// TwinCAT 3 PLC project AnalyticsPLC
// ProgramVersion: 3.1.4026.16
// libraries:
//   Tc2_EtherCAT, * (Beckhoff Automation GmbH)
//   Tc2_Standard, * (Beckhoff Automation GmbH)
//   Tc2_System, * (Beckhoff Automation GmbH)
//   Tc2_Utilities, * (Beckhoff Automation GmbH)
//   Tc3_Analytics, * (Beckhoff Automation GmbH)
//   Tc3_AnalyticsCommunication, * (Beckhoff Automation GmbH)
//   Tc3_EventLogger, * (Beckhoff Automation GmbH)
// project tree:
//   / AnalyticsTask.TcTTO, AnalyticsTask_C1.TcTTO, PlcTask.TcTTO
//   DUTs/Analytics/ Color.TcDUT, E_AnalysisComponents.TcDUT, E_DataSourceContext.TcDUT, E_DataSourceState.TcDUT, E_DTType.TcDUT, E_ScopeCommand.TcDUT, E_VirtualInput.TcDUT, Shapes.TcDUT, ST_AnalysisReset.TcDUT
//   DUTs/Analytics/HMI/Controls/ ST_HMI_C1_Ctrl1_Production_Quantity_Analysis.TcDUT, ST_HMI_C1_Ctrl2_OEE_Trend_Line.TcDUT, ST_HMI_C1_Ctrl3_Productivity_Interval.TcDUT, ST_HMI_C1_Ctrl4_Overall_Equipment_Effectiveness_OEE.TcDUT
//   DUTs/Analytics/HMI/DataSourcePage/ E_SourceType.TcDUT, ST_HMI_DataSourceConfig.TcDUT, ST_HMI_DataSourceCtrl.TcDUT, ST_HMI_DataSourceHist.TcDUT, ST_HMI_DataSourceHistInfo.TcDUT, ST_HMI_DataSourceHistRecordInfo.TcDUT, ST_HMI_InputSource.TcDUT, ST_HMI_InputSourceCtrl.TcDUT
//   DUTs/Analytics/HMI/ ST_HMI_C1_OEE_Status.TcDUT, ST_HMI_MapItem.TcDUT, ST_KeyValuePair.TcDUT
//   DUTs/Analytics/Results/ ST_Results.TcDUT
//   DUTs/Analytics/Sources/ ST_T1_Inputs.TcDUT
//   GVLs/ Analytics.TcGVL, AnalyticsHMI.TcGVL
//   POUs/Analytics/Analysis/ FB_Analysis.TcPOU
//   POUs/Analytics/Analysis/Networks/N01 OEEStatus/ FB_N1_OEEStatus.TcPOU
//   POUs/Analytics/Analysis/Networks/N01 OEEStatus/Modules/ FB_N1_M1_OverallEquipmentEffectivenessOEE.TcPOU, FB_N1_M2_ProductionModeTimingAnalysis.TcPOU, FB_N1_M3_OEETrendLine.TcPOU, FB_N1_M4_ProductionQuantityAnalysis.TcPOU, FB_N1_M5_ProductivityInterval.TcPOU
//   POUs/Analytics/ MAIN_Analytics.TcPOU, MAIN_Analytics_C1.TcPOU
//   POUs/Analytics/Sources/T1_InputSource/ FB_T1_InputSource.TcPOU
//   POUs/Analytics/Sources/[Interfaces]/ I_InputSource.TcIO, I_InputSourceHistorical.TcIO
//   POUs/Analytics/VirtualInputSources/C1_Configuration_1/ FB_V1_C1_VirtualInputSource.TcPOU
//   POUs/Analytics/VirtualInputSources/[Interfaces]/ I_V1_VirtualInputSource.TcIO, I_VirtualInputSource.TcIO
//   POUs/Analytics/[Helper]/Common/ FB_DataBuffer.TcPOU, FB_GetSampleIndex.TcPOU, FB_TcMessageSuccess.TcPOU, F_ANY_Negation.TcPOU, F_ARRAY_To_LREAL_ARRAY.TcPOU, F_HasContext.TcPOU, F_ToANY.TcPOU
//   POUs/Analytics/[Helper]/Convert Timestamp/ F_AlyTimestampToDCTimestruct.TcPOU, F_AlyTimestampToFileTime.TcPOU, F_AlyTimestampToLocalTime.TcPOU, F_DCTimestructToFileTime.TcPOU, F_FileTimeToDCTimestruct.TcPOU, F_RawTimeToDCTimestruct.TcPOU
//   POUs/Analytics/[Helper]/ F_SampleTimeCheck.TcPOU
//   POUs/ MAIN.TcPOU
// (motion and I/O tree: see PLC project unbenannt1)
// real-time tasks:
//   TASK PlcTask: cycle T#10ms, priority 20, ADS port 350
//   TASK PlcTask1: cycle T#10ms, priority 21, ADS port 351
//   TASK AnalyticsTask: cycle T#10ms, priority 1, ADS port 352
//   TASK AnalyticsTask_C1: cycle T#10ms, priority 22, ADS port 353
// variable links:

CONFIGURATION AnalyticsPLC
    RESOURCE PLC ON TwinCAT3
        TASK AnalyticsTask(INTERVAL := T#10ms, PRIORITY := 1);
        TASK AnalyticsTask_C1(INTERVAL := T#10ms, PRIORITY := 22);
        TASK PlcTask(INTERVAL := T#10ms, PRIORITY := 21);
        PROGRAM MAIN_Analytics WITH AnalyticsTask : MAIN_Analytics;
        PROGRAM MAIN_Analytics_C1 WITH AnalyticsTask_C1 : MAIN_Analytics_C1;
        PROGRAM MAIN WITH PlcTask : MAIN;
    END_RESOURCE
END_CONFIGURATION

// ---- DUTs/Analytics/Color.TcDUT
{attribute 'qualified_only'}
{attribute 'strict'}
TYPE Color : 
(
	White := 0,
	Black,
	Red,
	Green,
	Blue
) ;
END_TYPE

// ---- DUTs/Analytics/E_AnalysisComponents.TcDUT
{attribute 'qualified_only'}
{attribute 'strict'}
TYPE E_AnalysisComponents : 
(
	All := -1,
	N1_OEEStatus := 0,
	N1_M1_OverallEquipmentEffectivenessOEE := 1,
	N1_M2_ProductionModeTimingAnalysis := 2,
	N1_M3_OEETrendLine := 3,
	N1_M4_ProductionQuantityAnalysis := 4,
	N1_M5_ProductivityInterval := 5,
	V1_VirtualInputSource := 6
) ;
END_TYPE

// ---- DUTs/Analytics/E_DataSourceContext.TcDUT
{attribute 'qualified_only'}
TYPE E_DataSourceContext : 
(
	eContext_No := 0, //
	eContext_Unknown := 2#0000_0000_0000_0001_0000_0000_0000_0000, //Unknown - All contexts allowed
	eContext_10000 := 2#0000_0000_0000_0010_0000_0000_0000_0000, //10000 µs
	eContext_Reserve1 := 2#0000_0000_0000_0100_0000_0000_0000_0000, //Reserve
	eContext_Reserve2 := 2#0000_0000_0000_1000_0000_0000_0000_0000, //Reserve
	eContext_Reserve3 := 2#0000_0000_0001_0000_0000_0000_0000_0000, //Reserve
	eContext_Reserve4 := 2#0000_0000_0010_0000_0000_0000_0000_0000, //Reserve
	eContext_Reserve5 := 2#0000_0000_0100_0000_0000_0000_0000_0000, //Reserve
	eContext_Reserve6 := 2#0000_0000_1000_0000_0000_0000_0000_0000, //Reserve
	eContext_Reserve7 := 2#0000_0001_0000_0000_0000_0000_0000_0000, //Reserve
	eContext_Reserve8 := 2#0000_0010_0000_0000_0000_0000_0000_0000, //Reserve
	eContext_Reserve9 := 2#0000_0100_0000_0000_0000_0000_0000_0000, //Reserve
	eContext_Reserve10 := 2#0000_1000_0000_0000_0000_0000_0000_0000, //Reserve
	eContext_Reserve11 := 2#0001_0000_0000_0000_0000_0000_0000_0000, //Reserve
	eContext_Reserve12 := 2#0010_0000_0000_0000_0000_0000_0000_0000, //Reserve
	eContext_Reserve13 := 2#0100_0000_0000_0000_0000_0000_0000_0000, //Reserve
	eContext_Reserve14 := 2#1000_0000_0000_0000_0000_0000_0000_0000 //Reserve
) DWORD;
END_TYPE

// ---- DUTs/Analytics/E_DataSourceState.TcDUT
{attribute 'qualified_only'}
{attribute 'strict'}
TYPE E_DataSourceState : 
(
	eUnknown := 0,
	eNotConnected,
	eReceiveData,
	eReceiveData_Cancel,
	eReceiveData_Pause,
	eError,
	eReady,
	eWaitForData
) ;
END_TYPE

// ---- DUTs/Analytics/E_DTType.TcDUT
{attribute 'qualified_only'}
{attribute 'strict'}
TYPE E_DTType : 
(
	NotInitialized := 0,
	BOOL_,
	BYTE_,
	WORD_,
	DWORD_,
	SINT_,
	USINT_,
	INT_,
	UINT_,
	DINT_,
	UDINT_,
	LINT_,
	ULINT_,
	REAL_,
	LREAL_,
	LWORD_
) ;
END_TYPE

// ---- DUTs/Analytics/E_ScopeCommand.TcDUT
{attribute 'qualified_only'}
{attribute 'strict'}
TYPE E_ScopeCommand : 
(
	eDefault := 0,
	ePause,
	eStop
) ;
END_TYPE

// ---- DUTs/Analytics/E_VirtualInput.TcDUT
{attribute 'qualified_only'}
TYPE E_VirtualInput : 
(
	eContext_No := 0, //
	eContext_V1_VirtualInputSource := 2#0000_0000_0000_0000_0000_0000_0000_0001, //VirtualInputSource
	eContext_Vn_Reserve1 := 2#0000_0000_0000_0000_0000_0000_0000_0010, //Reserve
	eContext_Vn_Reserve2 := 2#0000_0000_0000_0000_0000_0000_0000_0100, //Reserve
	eContext_Vn_Reserve3 := 2#0000_0000_0000_0000_0000_0000_0000_1000, //Reserve
	eContext_Vn_Reserve4 := 2#0000_0000_0000_0000_0000_0000_0001_0000, //Reserve
	eContext_Vn_Reserve5 := 2#0000_0000_0000_0000_0000_0000_0010_0000, //Reserve
	eContext_Vn_Reserve6 := 2#0000_0000_0000_0000_0000_0000_0100_0000, //Reserve
	eContext_Vn_Reserve7 := 2#0000_0000_0000_0000_0000_0000_1000_0000, //Reserve
	eContext_Vn_Reserve8 := 2#0000_0000_0000_0000_0000_0001_0000_0000, //Reserve
	eContext_Vn_Reserve9 := 2#0000_0000_0000_0000_0000_0010_0000_0000, //Reserve
	eContext_Vn_Reserve10 := 2#0000_0000_0000_0000_0000_0100_0000_0000, //Reserve
	eContext_Vn_Reserve11 := 2#0000_0000_0000_0000_0000_1000_0000_0000, //Reserve
	eContext_Vn_Reserve12 := 2#0000_0000_0000_0000_0001_0000_0000_0000, //Reserve
	eContext_Vn_Reserve13 := 2#0000_0000_0000_0000_0010_0000_0000_0000, //Reserve
	eContext_Vn_Reserve14 := 2#0000_0000_0000_0000_0100_0000_0000_0000, //Reserve
	eContext_Vn_Reserve15 := 2#0000_0000_0000_0000_1000_0000_0000_0000 //Reserve
) DWORD;
END_TYPE

// ---- DUTs/Analytics/HMI/Controls/ST_HMI_C1_Ctrl1_Production_Quantity_Analysis.TcDUT
TYPE ST_HMI_C1_Ctrl1_Production_Quantity_Analysis : 
STRUCT
	//Production Quantity Analysis
	bTrigReconfigure: BOOL;
	fM4_nCyclesElapsed: LREAL; //Elapsed (Values)
	fM4_nCyclesRemaining: LREAL; //Remaining (Values)
END_STRUCT
END_TYPE

// ---- DUTs/Analytics/HMI/Controls/ST_HMI_C1_Ctrl2_OEE_Trend_Line.TcDUT
TYPE ST_HMI_C1_Ctrl2_OEE_Trend_Line : 
STRUCT
	//OEE Trend Line
	bTrigReconfigure: BOOL;
	aM3_aTrendData: ARRAY [1..4] OF ARRAY [1..10080] OF LREAL; //Raw Data
	tM3_fbLastValue: DCTIMESTRUCT; //Last Value Timestamp
	nM3_nCountValues: UDINT; //Counted Values
	aM3_aChannelNames: ARRAY [0..3] OF STRING(255); //Display Names
END_STRUCT
END_TYPE

// ---- DUTs/Analytics/HMI/Controls/ST_HMI_C1_Ctrl3_Productivity_Interval.TcDUT
TYPE ST_HMI_C1_Ctrl3_Productivity_Interval : 
STRUCT
	//Productivity Interval
	bTrigReconfigure: BOOL;
	fM5_nProducedInInterval: LREAL; //Produced Pieces
	fM5_nRemainingInInterval: LREAL; //Remaining Pieces
	tM5_fbElapsedTime: ST_ALY_TimeSpan; //Elapsed Time
	tM5_fbRemainingTime: ST_ALY_TimeSpan; //Remaining Time
	fM5_fCurrentProductivity: LREAL; //Current Productivity
	fM5_fExpectedProductivity: LREAL; //Expected Productivity
END_STRUCT
END_TYPE

// ---- DUTs/Analytics/HMI/Controls/ST_HMI_C1_Ctrl4_Overall_Equipment_Effectiveness_OEE.TcDUT
TYPE ST_HMI_C1_Ctrl4_Overall_Equipment_Effectiveness_OEE : 
STRUCT
	//Overall Equipment Effectiveness (OEE)
	bTrigReconfigure: BOOL;
	fM1_fOEE: LREAL; //Overall equipment effectiveness (OEE)
	fM1_fAvailability: LREAL; //Availability
	fM1_fPerformance: LREAL; //Performance
	fM1_fQuality: LREAL; //Quality
	fM1_fThresholdLevelOkWarning: LREAL; //Level Ok / Warning
	fM1_fThresholdLevelWarningAlarm: LREAL; //Level Warning / Alarm
	eM1_eOeeClass: E_ALY_Classification_3Cls; //OEE Classification
END_STRUCT
END_TYPE

// ---- DUTs/Analytics/HMI/DataSourcePage/E_SourceType.TcDUT
{attribute 'qualified_only'}
{attribute 'strict'}
TYPE E_SourceType : 
(
	eLive := 0,
	eHistMQTT,
	eHistFile
) ;
END_TYPE

// ---- DUTs/Analytics/HMI/DataSourcePage/ST_HMI_DataSourceConfig.TcDUT
TYPE ST_HMI_DataSourceConfig : 
STRUCT
	nID: DINT;
	sDisplayName: WSTRING(80);
	eConfigType: E_SourceType;
	aInputSources: ARRAY [0..0] OF ST_HMI_InputSource;
END_STRUCT
END_TYPE

// ---- DUTs/Analytics/HMI/DataSourcePage/ST_HMI_DataSourceCtrl.TcDUT
TYPE ST_HMI_DataSourceCtrl : 
STRUCT
	nActiveConfigurationIdx: INT;
	
	aInputSourceCtrls: ARRAY [0..0] OF ST_HMI_InputSourceCtrl;
	
	bStart: BOOL;
	bCancel: BOOL;
	bPause: BOOL;
	bReset: BOOL;
	
	bUpdateRecordList: BOOL;
END_STRUCT
END_TYPE

// ---- DUTs/Analytics/HMI/DataSourcePage/ST_HMI_DataSourceHist.TcDUT
TYPE ST_HMI_DataSourceHist : 
STRUCT
	nCurrentRecordID: DINT;
	stSourceInfo: ST_HMI_DataSourceHistInfo;
	nRecordCount: DINT;
	aRecords: ARRAY [0..255] OF ST_HMI_DataSourceHistRecordInfo;
END_STRUCT
END_TYPE

// ---- DUTs/Analytics/HMI/DataSourcePage/ST_HMI_DataSourceHistInfo.TcDUT
TYPE ST_HMI_DataSourceHistInfo : 
STRUCT
	sSPGuid: GUID;
	sAlyFilePath: STRING(255);
	sSourceType: STRING(80);
	sTopic: STRING(255);
	sLayoutID: GUID;
END_STRUCT
END_TYPE

// ---- DUTs/Analytics/HMI/DataSourcePage/ST_HMI_DataSourceHistRecordInfo.TcDUT
TYPE ST_HMI_DataSourceHistRecordInfo : 
STRUCT
	nID: DINT;
	sName: WSTRING(80);
	sDisplayName: WSTRING(80);
	dtRecordStart: DCTIMESTRUCT;
	dtRecordEnd: DCTIMESTRUCT;
	dtSelectedRangeStart: DCTIMESTRUCT;
	dtSelectedRangeEnd: DCTIMESTRUCT;
END_STRUCT
END_TYPE

// ---- DUTs/Analytics/HMI/DataSourcePage/ST_HMI_InputSource.TcDUT
TYPE ST_HMI_InputSource : 
STRUCT
	nID: DINT;
	sDisplayName: WSTRING(80);
	
	sStreamSystemID: GUID;
	sTopic: STRING(255);
	
	eSourceType: E_SourceType;;
	eState: E_DataSourceState;;
	dtTimestamp: DCTIMESTRUCT;
	
	stHist: ST_HMI_DataSourceHist;
END_STRUCT
END_TYPE

// ---- DUTs/Analytics/HMI/DataSourcePage/ST_HMI_InputSourceCtrl.TcDUT
TYPE ST_HMI_InputSourceCtrl : 
STRUCT
	nActiveRecordIdx: INT;
	
	dtSelectedRangeStart: DCTIMESTRUCT;
	dtSelectedRangeEnd: DCTIMESTRUCT;
	
	bStart: BOOL;
	bCancel: BOOL;
	bPause: BOOL;
	bReset: BOOL;
END_STRUCT
END_TYPE

// ---- DUTs/Analytics/HMI/ST_HMI_C1_OEE_Status.TcDUT
TYPE ST_HMI_C1_OEE_Status : 
STRUCT
	stHMI_C1_Ctrl4_Overall_Equipment_Effectiveness_OEE: ST_HMI_C1_Ctrl4_Overall_Equipment_Effectiveness_OEE;
	
	stHMI_C1_Ctrl2_OEE_Trend_Line: ST_HMI_C1_Ctrl2_OEE_Trend_Line;
	
	stHMI_C1_Ctrl1_Production_Quantity_Analysis: ST_HMI_C1_Ctrl1_Production_Quantity_Analysis;
	
	stHMI_C1_Ctrl3_Productivity_Interval: ST_HMI_C1_Ctrl3_Productivity_Interval;
END_STRUCT
END_TYPE

// ---- DUTs/Analytics/HMI/ST_HMI_MapItem.TcDUT
TYPE ST_HMI_MapItem : 
STRUCT
	sName: WSTRING(127);
	sDescription: WSTRING(127);
	sPosition: WSTRING(127);
	nStatus: INT;
END_STRUCT
END_TYPE

// ---- DUTs/Analytics/HMI/ST_KeyValuePair.TcDUT
TYPE ST_KeyValuePair : 
STRUCT
	sKey: WSTRING(127);
	sValue: STRING(255);
END_STRUCT
END_TYPE

// ---- DUTs/Analytics/Results/ST_Results.TcDUT
TYPE ST_Results : 
STRUCT
END_STRUCT
END_TYPE

// ---- DUTs/Analytics/Shapes.TcDUT
{attribute 'qualified_only'}
{attribute 'strict'}
TYPE Shapes : 
(
	Rectangle := 0,
	Triangle,
	Pentagon,
	Hexagon,
	Circle
) ;
END_TYPE

// ---- DUTs/Analytics/Sources/ST_T1_Inputs.TcDUT
TYPE ST_T1_Inputs : 
STRUCT
	bGlobalVariables_bProductionMode: BOOL; //GlobalVariables.bProductionMode
	nGlobalVariables_lScheduledTime: LINT; //GlobalVariables.lScheduledTime
	nGlobalVariables_uProcessedCount: ULINT; //GlobalVariables.uProcessedCount
	nGlobalVariables_nVisuProductCommand: DINT; //GlobalVariables.nVisuProductCommand
	nGlobalVariables_uDefectiveCount: ULINT; //GlobalVariables.uDefectiveCount
	nGlobalVariables_lStartTime: LWORD; //GlobalVariables.lStartTime
	nGlobalVariables_lStopTime: LWORD; //GlobalVariables.lStopTime
	bGlobalVariables_bConfigure: BOOL; //GlobalVariables.bConfigure
	bGlobalVariables_bReset: BOOL; //GlobalVariables.bReset
	bGlobalVariables_bTest: BOOL; //GlobalVariables.bTest
	nGlobalVariables_uTotalCount: ULINT; //GlobalVariables.uTotalCount
END_STRUCT
END_TYPE

// ---- DUTs/Analytics/ST_AnalysisReset.TcDUT
TYPE ST_AnalysisReset : 
STRUCT
	eResetComponent: E_AnalysisComponents := E_AnalysisComponents.All;
	bResetExecute: BOOL;
END_STRUCT
END_TYPE

// ---- GVLs/Analytics.TcGVL
{attribute 'qualified_only'}
VAR_GLOBAL
	//DataSources
	//Live:
	fbT1_InputSource: FB_T1_InputSource;
	//Historical:
	//Empty:
	
	fbT1_IecCriticalSection: FB_IecCriticalSection;
	
	//Historical DataSource parameter
	nHistMaxInputBuffer: UDINT := 100;
	nHistMaxSampleCount: UDINT := 100;
	
	stReset: ST_AnalysisReset;
	
	//Scope ADS Push Target NetID
	sScopeServerNetID: T_AmsNetID := '10.123.65.55.1.1';
END_VAR

// ---- GVLs/AnalyticsHMI.TcGVL
{attribute 'qualified_only'}
VAR_GLOBAL
	//Switch between historical and live data
	stHMI_DataSourceCtrl: ST_HMI_DataSourceCtrl;
	stHMI_DataSourceConfig: ARRAY [0..0] OF ST_HMI_DataSourceConfig := [ 
																	( nID:= 1, sDisplayName:= "Configuration 1", eConfigType:= E_SourceType.eLive, 
																		aInputSources:= [ 
																			( nID:= 1, sDisplayName:= "1aa71777-6a15-92b4-38b4-ceb9ef9aa20f", sStreamSystemID:= STRING_TO_GUID('1aa71777-6a15-92b4-38b4-ceb9ef9aa20f'), 
																				sTopic:= 'PackMLDemo/PlcStream1', eSourceType:= E_SourceType.eLive, eState:= E_DataSourceState.eUnknown ) ] ) ];
	
	//Reset
	bN1_OEEStatus_Reset: BOOL;
	bN1_M1_OverallEquipmentEffectivenessOEE_Reset: BOOL;
	bN1_M2_ProductionModeTimingAnalysis_Reset: BOOL;
	bN1_M3_OEETrendLine_Reset: BOOL;
	bN1_M4_ProductionQuantityAnalysis_Reset: BOOL;
	bN1_M5_ProductivityInterval_Reset: BOOL;
	
	//Virtual Inputs
	bV1_bProductionMode: BOOL;
	nV1_lScheduledTime: LINT;
	nV1_uDefectiveCount: ULINT;
	nV1_lStartTime: LWORD;
	nV1_lStopTime: LWORD;
	bV1_bConfigure: BOOL;
	bV1_bReset: BOOL;
	bV1_bTest: BOOL;
	nV1_uTotalCount: ULINT;
	
	//HMI Structs
	stHMI_C1_OEE_Status: ST_HMI_C1_OEE_Status;
	
	//HMI Map Items
	aMapItems: ARRAY [0..0] OF ST_HMI_MapItem := [(sName:="1aa71777-6a15-92b4-38b4-ceb9ef9aa20f", sDescription:="", sPosition:="3 International Business Park, #05-07/08 Nordic European Centre, Singapore 609927", nStatus:= 0)];
END_VAR
VAR_GLOBAL CONSTANT
	nInstanceId: ULINT := 12860370723493188529;
END_VAR

// ---- POUs/Analytics/Sources/[Interfaces]/I_InputSource.TcIO
INTERFACE I_InputSource

METHOD AddClient : BOOL
VAR_OUTPUT
	nClientID: LWORD;
END_VAR
END_METHOD

METHOD Call : BOOL
END_METHOD

METHOD ClientDone : BOOL
VAR_INPUT
	nClientID: LWORD;
END_VAR
END_METHOD

METHOD GetData : BOOL
VAR_INPUT
	nElement: UDINT;
	pInputs: PVOID;
	nInputsSize: UDINT;
END_VAR
VAR_OUTPUT
	nTimestamp: ULINT;
	nContext: DWORD;
END_VAR
END_METHOD

METHOD NewDataAvailable : BOOL
VAR_INPUT
	nLastDataHandle: ULINT;
END_VAR
END_METHOD

PROPERTY eDataState : E_DataSourceState
GET
END_GET
END_PROPERTY

PROPERTY bReadNewData : BOOL
GET
END_GET
END_PROPERTY

PROPERTY nDataHandle : ULINT
GET
END_GET
END_PROPERTY

PROPERTY nElements : UDINT
GET
END_GET
END_PROPERTY

END_INTERFACE

// ---- POUs/Analytics/Sources/[Interfaces]/I_InputSourceHistorical.TcIO
INTERFACE I_InputSourceHistorical EXTENDS I_InputSource

METHOD HistoricalCtrl : BOOL
VAR_INPUT
	stCtrl: REFERENCE TO ST_HMI_InputSourceCtrl;
	stHistStreamInfo: REFERENCE TO ST_HMI_DataSourceHist;
	stRecordInfo: REFERENCE TO ST_HMI_DataSourceHistRecordInfo;
END_VAR
END_METHOD

METHOD UpdateRecordList : BOOL
VAR_INPUT
	sStreamSystemID: GUID;
	stHistStreamInfo: REFERENCE TO ST_HMI_DataSourceHist;
END_VAR
END_METHOD

PROPERTY bCtrlChanged : BOOL
GET
END_GET
END_PROPERTY

END_INTERFACE

// ---- POUs/Analytics/VirtualInputSources/[Interfaces]/I_V1_VirtualInputSource.TcIO
INTERFACE I_V1_VirtualInputSource EXTENDS I_VirtualInputSource

PROPERTY nV1_TimeLine : ULINT
GET
END_GET
END_PROPERTY

PROPERTY bV1_bProductionMode : BOOL
GET
END_GET
END_PROPERTY

PROPERTY nV1_lScheduledTime : LINT
GET
END_GET
END_PROPERTY

PROPERTY nV1_uDefectiveCount : ULINT
GET
END_GET
END_PROPERTY

PROPERTY nV1_lStartTime : LWORD
GET
END_GET
END_PROPERTY

PROPERTY nV1_lStopTime : LWORD
GET
END_GET
END_PROPERTY

PROPERTY bV1_bConfigure : BOOL
GET
END_GET
END_PROPERTY

PROPERTY bV1_bReset : BOOL
GET
END_GET
END_PROPERTY

PROPERTY bV1_bTest : BOOL
GET
END_GET
END_PROPERTY

PROPERTY nV1_uTotalCount : ULINT
GET
END_GET
END_PROPERTY

END_INTERFACE

// ---- POUs/Analytics/VirtualInputSources/[Interfaces]/I_VirtualInputSource.TcIO
INTERFACE I_VirtualInputSource

METHOD Done : BOOL
END_METHOD

METHOD NextData : BOOL
VAR_INPUT
	nMaxOversampling: UDINT;
END_VAR
END_METHOD

METHOD SourceSync : BOOL
END_METHOD

PROPERTY bEndOfData : BOOL
GET
END_GET
END_PROPERTY

PROPERTY dtTimestamp : DCTIMESTRUCT
GET
END_GET
END_PROPERTY

PROPERTY nContext : DWORD
GET
END_GET
END_PROPERTY

PROPERTY nDataHandle : ULINT
GET
END_GET
END_PROPERTY

PROPERTY tTimestamp : ULINT
GET
END_GET
END_PROPERTY

PROPERTY nMaxOversamplingFactor : UDINT
GET
END_GET
END_PROPERTY

PROPERTY eSourceState : E_DataSourceState
GET
END_GET
END_PROPERTY

END_INTERFACE

// ---- POUs/Analytics/MAIN_Analytics.TcPOU
PROGRAM MAIN_Analytics
VAR
END_VAR


//Reset Analytics Components
A_Reset();

CASE AnalyticsHMI.stHMI_DataSourceCtrl.nActiveConfigurationIdx OF
	0:

		//Reset
		MAIN_Analytics_C1.A_Reset(stReset := Analytics.stReset);

		//Map to HMI
		MAIN_Analytics_C1.A_MapToHMI();
END_CASE


//Call DataSource FBs
IF Analytics.fbT1_InputSource.bReadNewData THEN
	Analytics.fbT1_InputSource.Call();
END_IF

ACTION A_Reset:

IF AnalyticsHMI.bN1_OEEStatus_Reset THEN
	Analytics.stReset.eResetComponent:= E_AnalysisComponents.N1_OEEStatus;
	Analytics.stReset.bResetExecute:= TRUE;
	AnalyticsHMI.bN1_OEEStatus_Reset:= FALSE;
END_IF

IF AnalyticsHMI.bN1_M1_OverallEquipmentEffectivenessOEE_Reset THEN
	Analytics.stReset.eResetComponent:= E_AnalysisComponents.N1_M1_OverallEquipmentEffectivenessOEE;
	Analytics.stReset.bResetExecute:= TRUE;
	AnalyticsHMI.bN1_M1_OverallEquipmentEffectivenessOEE_Reset:= FALSE;
END_IF

IF AnalyticsHMI.bN1_M2_ProductionModeTimingAnalysis_Reset THEN
	Analytics.stReset.eResetComponent:= E_AnalysisComponents.N1_M2_ProductionModeTimingAnalysis;
	Analytics.stReset.bResetExecute:= TRUE;
	AnalyticsHMI.bN1_M2_ProductionModeTimingAnalysis_Reset:= FALSE;
END_IF

IF AnalyticsHMI.bN1_M3_OEETrendLine_Reset THEN
	Analytics.stReset.eResetComponent:= E_AnalysisComponents.N1_M3_OEETrendLine;
	Analytics.stReset.bResetExecute:= TRUE;
	AnalyticsHMI.bN1_M3_OEETrendLine_Reset:= FALSE;
END_IF

IF AnalyticsHMI.bN1_M4_ProductionQuantityAnalysis_Reset THEN
	Analytics.stReset.eResetComponent:= E_AnalysisComponents.N1_M4_ProductionQuantityAnalysis;
	Analytics.stReset.bResetExecute:= TRUE;
	AnalyticsHMI.bN1_M4_ProductionQuantityAnalysis_Reset:= FALSE;
END_IF

IF AnalyticsHMI.bN1_M5_ProductivityInterval_Reset THEN
	Analytics.stReset.eResetComponent:= E_AnalysisComponents.N1_M5_ProductivityInterval;
	Analytics.stReset.bResetExecute:= TRUE;
	AnalyticsHMI.bN1_M5_ProductivityInterval_Reset:= FALSE;
END_IF
END_ACTION

END_PROGRAM

// ---- POUs/Analytics/MAIN_Analytics_C1.TcPOU
PROGRAM MAIN_Analytics_C1
VAR_INPUT
	stReset: ST_AnalysisReset;
END_VAR
VAR_OUTPUT
	bError: BOOL;
	ipTcResult: I_TcMessage;
END_VAR
VAR
	nHMIUpdateState: INT;
	bHMIReinit: BOOL := TRUE;
	bHMIResetReinit: BOOL;
	bHMIReinitDone: BOOL;
	
	fbV1_C1_VirtualInputSource: FB_V1_C1_VirtualInputSource(fbSource:= Analytics.fbT1_InputSource);
	
	fbAnalysis: FB_Analysis := ( nConfigurationID:= 1, 
								ipVirtualInputSource:= fbV1_C1_VirtualInputSource );
END_VAR

A_Reset();

fbV1_C1_VirtualInputSource.SourceSync();

IF NOT fbV1_C1_VirtualInputSource.bEndOfData THEN

	WHILE NOT fbV1_C1_VirtualInputSource.bEndOfData DO

		fbV1_C1_VirtualInputSource.NextData(1);

		fbAnalysis.Call();

	END_WHILE

ELSE
	fbAnalysis.Call();
END_IF

fbV1_C1_VirtualInputSource.Done();

//Error Handling
bError:= fbAnalysis.bError;
ipTcResult:= fbAnalysis.ipTcResult;


//Map HMI Current Timestamp
AnalyticsHMI.stHMI_DataSourceConfig[0].aInputSources[0].eState:= fbV1_C1_VirtualInputSource.fbInputSource.eDataState;
AnalyticsHMI.stHMI_DataSourceConfig[0].aInputSources[0].dtTimestamp:= fbV1_C1_VirtualInputSource.dtTimestamp;

ACTION A_Reset:

//Reset Analytics Components
fbAnalysis.Reset(stReset);

Analytics.stReset.bResetExecute:= FALSE;
END_ACTION

ACTION A_MapToHMI:

//Map In-/Outputs of the Analysis to HMI Structs
CASE nHMIUpdateState OF
	0:
		bHMIReinit:= bHMIReinit OR fbAnalysis.GetHMIValues(1, ADR(AnalyticsHMI.stHMI_C1_OEE_Status));
		bHMIReinitDone:= fbAnalysis.SetHMIValues(1, ADR(AnalyticsHMI.stHMI_C1_OEE_Status), bHMIReinit);
		nHMIUpdateState:= 1;
	1:
		AnalyticsHMI.bV1_bProductionMode:= fbV1_C1_VirtualInputSource.bV1_bProductionMode;
		AnalyticsHMI.nV1_lScheduledTime:= fbV1_C1_VirtualInputSource.nV1_lScheduledTime;
		AnalyticsHMI.nV1_uDefectiveCount:= fbV1_C1_VirtualInputSource.nV1_uDefectiveCount;
		AnalyticsHMI.nV1_lStartTime:= fbV1_C1_VirtualInputSource.nV1_lStartTime;
		AnalyticsHMI.nV1_lStopTime:= fbV1_C1_VirtualInputSource.nV1_lStopTime;
		AnalyticsHMI.bV1_bConfigure:= fbV1_C1_VirtualInputSource.bV1_bConfigure;
		AnalyticsHMI.bV1_bReset:= fbV1_C1_VirtualInputSource.bV1_bReset;
		AnalyticsHMI.bV1_bTest:= fbV1_C1_VirtualInputSource.bV1_bTest;
		AnalyticsHMI.nV1_uTotalCount:= fbV1_C1_VirtualInputSource.nV1_uTotalCount;
		nHMIUpdateState:= 2;
	2:
		IF bHMIResetReinit THEN
			bHMIResetReinit:= FALSE;
			bHMIReinit:= FALSE;
		END_IF

		IF bHMIReinitDone THEN
			bHMIResetReinit:= TRUE;
		END_IF

		nHMIUpdateState:= 0;
END_CASE
END_ACTION

END_PROGRAM

// ---- POUs/Analytics/VirtualInputSources/C1_Configuration_1/FB_V1_C1_VirtualInputSource.TcPOU
FUNCTION_BLOCK FB_V1_C1_VirtualInputSource IMPLEMENTS I_VirtualInputSource, I_V1_VirtualInputSource
VAR
	_fbSource: I_InputSource;
	
	_nSourceClientID: LWORD;
	_nDataHandle: ULINT;
	_nElements: UDINT;
	
	_nSelectedElement: UDINT;
	_nSelectedOversample: UDINT;
	
	_nMaxOversamplingFactor: UDINT := 1;
	
	_nContext: DWORD;
	_stInputs: ST_T1_Inputs;
	
	_nTimestamp: ULINT;
END_VAR

METHOD Done : BOOL
VAR
END_VAR
IF bEndOfData AND _nElements > 0 THEN
	_nElements:= 0;
	_fbSource.ClientDone(_nSourceClientID);
END_IF

_nContext:= 0;
END_METHOD

METHOD NextData : BOOL
VAR_INPUT
	nMaxOversampling: UDINT;
END_VAR
VAR
END_VAR
IF _nElements > 0 AND NOT bEndOfData THEN

	_nSelectedOversample:= _nSelectedOversample + 1;
	IF _nSelectedOversample > nMaxOversampling OR _nSelectedElement = 0 THEN
		_nSelectedElement:= _nSelectedElement + 1;
		_nSelectedOversample:= 1;
	END_IF

	NextData:= _fbSource.GetData(_nSelectedElement, ADR(_stInputs), SIZEOF(_stInputs), nTimestamp=>_nTimestamp, nContext=>_nContext);
	_nContext:= _nContext OR E_VirtualInput.eContext_V1_VirtualInputSource;
END_IF
END_METHOD

METHOD SourceSync : BOOL
VAR
END_VAR
IF _fbSource.NewDataAvailable(_nDataHandle) THEN
	_nDataHandle:= _fbSource.nDataHandle;
	_nElements:= _fbSource.nElements;

	_nSelectedElement:= 0;
	_nSelectedOversample:= 0;
END_IF
END_METHOD

METHOD FB_init : BOOL
VAR_INPUT
	bInitRetains: BOOL; // if TRUE, the retain variables are initialized (warm start / cold start)
	bInCopyCode: BOOL; // if TRUE, the instance afterwards gets moved into the copy code (online change)
	fbSource: I_InputSource;
END_VAR
VAR
END_VAR
IF NOT bInCopyCode THEN
	fbSource.AddClient(nClientID=>_nSourceClientID);
	_fbSource:= fbSource;
END_IF
END_METHOD

PROPERTY bEndOfData : BOOL
GET
bEndOfData:= _nElements = 0 OR (_nSelectedElement >= _nElements AND _nSelectedOversample >= _nMaxOversamplingFactor);
END_GET
END_PROPERTY

PROPERTY dtTimestamp : DCTIMESTRUCT
GET
dtTimestamp:= F_AlyTimestampToDCTimestruct(_nTimestamp);
END_GET
END_PROPERTY

PROPERTY nContext : DWORD
GET
nContext:= _nContext;
END_GET
END_PROPERTY

PROPERTY nDataHandle : ULINT
GET
nDataHandle:= _nDataHandle;
END_GET
END_PROPERTY

PROPERTY tTimestamp : ULINT
GET
tTimestamp:= _nTimestamp;
END_GET
END_PROPERTY

PROPERTY nMaxOversamplingFactor : UDINT
GET
nMaxOversamplingFactor:= _nMaxOversamplingFactor;
END_GET
END_PROPERTY

PROPERTY eSourceState : E_DataSourceState
GET
eSourceState:= _fbSource.eDataState;
END_GET
END_PROPERTY

PROPERTY nV1_TimeLine : ULINT
GET
//Timeline Value
nV1_TimeLine:= _nTimestamp;
END_GET
END_PROPERTY

PROPERTY bV1_bProductionMode : BOOL
GET
bV1_bProductionMode:= _stInputs.bGlobalVariables_bProductionMode;
END_GET
END_PROPERTY

PROPERTY nV1_lScheduledTime : LINT
GET
nV1_lScheduledTime:= _stInputs.nGlobalVariables_lScheduledTime;
END_GET
END_PROPERTY

PROPERTY nV1_uDefectiveCount : ULINT
GET
nV1_uDefectiveCount:= _stInputs.nGlobalVariables_uDefectiveCount;
END_GET
END_PROPERTY

PROPERTY nV1_lStartTime : LWORD
GET
nV1_lStartTime:= _stInputs.nGlobalVariables_lStartTime;
END_GET
END_PROPERTY

PROPERTY nV1_lStopTime : LWORD
GET
nV1_lStopTime:= _stInputs.nGlobalVariables_lStopTime;
END_GET
END_PROPERTY

PROPERTY bV1_bConfigure : BOOL
GET
bV1_bConfigure:= _stInputs.bGlobalVariables_bConfigure;
END_GET
END_PROPERTY

PROPERTY bV1_bReset : BOOL
GET
bV1_bReset:= _stInputs.bGlobalVariables_bReset;
END_GET
END_PROPERTY

PROPERTY bV1_bTest : BOOL
GET
bV1_bTest:= _stInputs.bGlobalVariables_bTest;
END_GET
END_PROPERTY

PROPERTY nV1_uTotalCount : ULINT
GET
nV1_uTotalCount:= _stInputs.nGlobalVariables_uTotalCount;
END_GET
END_PROPERTY

PROPERTY fbInputSource : I_InputSource
GET
fbInputSource:= _fbSource;
END_GET
END_PROPERTY

END_FUNCTION_BLOCK

// ---- POUs/Analytics/[Helper]/Convert Timestamp/F_AlyTimestampToDCTimestruct.TcPOU
FUNCTION F_AlyTimestampToDCTimestruct : DCTIMESTRUCT
VAR_INPUT
	tTimestamp: ULINT;
END_VAR
VAR
	tFileTime: T_FILETIME;
	newDCTime: T_DCTIME64;
	
	fbToLocal: FB_FileTimeToTzSpecificLocalTime;
	//Malay Peninsula Daylight Time
	//(UTC+08:00) Kuala Lumpur, Singapore
	tzInfo: ST_TimeZoneInformation := (bias := -480);
END_VAR

tFileTime:= DCTIME64_TO_Filetime(tTimestamp);
fbToLocal(in:= tFileTime, tzInfo:= tzInfo);
newDCTime:= FILETIME_TO_DCTIME64(fbToLocal.out);

F_AlyTimestampToDCTimestruct:= DCTIME64_TO_DCTIMESTRUCT(newDCTime);

END_FUNCTION

// ---- POUs/Analytics/Analysis/FB_Analysis.TcPOU
FUNCTION_BLOCK FB_Analysis
VAR_INPUT
	nConfigurationID: INT;
	ipVirtualInputSource: I_V1_VirtualInputSource;
	
END_VAR
VAR_OUTPUT
	bError: BOOL;
	ipTcResult: I_TcMessage := fbTcMsgSuccess;
END_VAR
VAR
	fbTcMsgSuccess: FB_TcMessageSuccess;
	
	R_TRIG_Reset: R_TRIG;
	bResetBusy: BOOL;
	
	fbN1_OEEStatus: FB_N1_OEEStatus;
END_VAR

METHOD Reset : BOOL
VAR_IN_OUT
	stReset: ST_AnalysisReset;
END_VAR
VAR
END_VAR

R_TRIG_Reset(CLK:= stReset.bResetExecute);
IF R_TRIG_Reset.Q OR bResetBusy THEN
	bResetBusy:= TRUE;

	CASE stReset.eResetComponent OF
		E_AnalysisComponents.All:
			bResetBusy:= bResetBusy AND fbN1_OEEStatus.Reset();
		E_AnalysisComponents.N1_OEEStatus:
			bResetBusy:= bResetBusy AND fbN1_OEEStatus.Reset();
		E_AnalysisComponents.N1_M1_OverallEquipmentEffectivenessOEE:
			bResetBusy:= bResetBusy AND fbN1_OEEStatus.fbM1_OverallEquipmentEffectivenessOEE.Reset();
		E_AnalysisComponents.N1_M2_ProductionModeTimingAnalysis:
			bResetBusy:= bResetBusy AND fbN1_OEEStatus.fbM2_ProductionModeTimingAnalysis.Reset();
		E_AnalysisComponents.N1_M3_OEETrendLine:
			bResetBusy:= bResetBusy AND fbN1_OEEStatus.fbM3_OEETrendLine.Reset();
		E_AnalysisComponents.N1_M4_ProductionQuantityAnalysis:
			bResetBusy:= bResetBusy AND fbN1_OEEStatus.fbM4_ProductionQuantityAnalysis.Reset();
		E_AnalysisComponents.N1_M5_ProductivityInterval:
			bResetBusy:= bResetBusy AND fbN1_OEEStatus.fbM5_ProductivityInterval.Reset();
		E_AnalysisComponents.V1_VirtualInputSource:
			bResetBusy:= bResetBusy AND fbN1_OEEStatus.fbM1_OverallEquipmentEffectivenessOEE.Reset();
			bResetBusy:= bResetBusy AND fbN1_OEEStatus.fbM2_ProductionModeTimingAnalysis.Reset();
			bResetBusy:= bResetBusy AND fbN1_OEEStatus.fbM3_OEETrendLine.Reset();
			bResetBusy:= bResetBusy AND fbN1_OEEStatus.fbM4_ProductionQuantityAnalysis.Reset();
			bResetBusy:= bResetBusy AND fbN1_OEEStatus.fbM5_ProductivityInterval.Reset();
	END_CASE

	bResetBusy:= NOT bResetBusy;

	stReset.bResetExecute:= bResetBusy;
END_IF
END_METHOD

METHOD Call : BOOL
VAR
END_VAR

//Analytics Network "OEEStatus" with ID: 1
fbN1_OEEStatus.Call(THIS);


//Error Handling
IF fbN1_OEEStatus.bError THEN
	bError:= TRUE;
	ipTcResult:= fbN1_OEEStatus.ipTcResult;
ELSE
	bError:= FALSE;
	ipTcResult:= fbTcMsgSuccess;
END_IF
END_METHOD

METHOD SetHMIValues : BOOL
VAR_INPUT
	nContentID: DINT;
	pContent: PVOID;
	bHMIReinit: BOOL;
END_VAR
VAR
END_VAR

CASE nContentID OF
	1:
		SetHMIValues:= fbN1_OEEStatus.fbM1_OverallEquipmentEffectivenessOEE.SetHMI(1, pContent, bHMIReinit);
		SetHMIValues:= SetHMIValues AND fbN1_OEEStatus.fbM3_OEETrendLine.SetHMI(1, pContent, bHMIReinit);
		SetHMIValues:= SetHMIValues AND fbN1_OEEStatus.fbM4_ProductionQuantityAnalysis.SetHMI(1, pContent, bHMIReinit);
		SetHMIValues:= SetHMIValues AND fbN1_OEEStatus.fbM5_ProductivityInterval.SetHMI(1, pContent, bHMIReinit);
END_CASE
END_METHOD

METHOD GetHMIValues : BOOL
VAR_INPUT
	nContentID: DINT;
	pContent: PVOID;
END_VAR
VAR
END_VAR

CASE nContentID OF
	1:
		GetHMIValues:= fbN1_OEEStatus.fbM1_OverallEquipmentEffectivenessOEE.GetHMI(1, pContent);
		GetHMIValues:= GetHMIValues OR fbN1_OEEStatus.fbM3_OEETrendLine.GetHMI(1, pContent);
END_CASE
END_METHOD

PROPERTY nContext : DWORD
GET

nContext:= 0;
IF ipVirtualInputSource <> 0 THEN
	nContext:= ipVirtualInputSource.nContext;
END_IF
END_GET
END_PROPERTY

END_FUNCTION_BLOCK

// ---- POUs/Analytics/[Helper]/Common/FB_TcMessageSuccess.TcPOU
FUNCTION_BLOCK FB_TcMessageSuccess EXTENDS FB_TcMessage
VAR
END_VAR

METHOD FB_init : BOOL
VAR_INPUT
	bInitRetains: BOOL; // if TRUE, the retain variables are initialized (warm start / cold start)
	bInCopyCode: BOOL; // if TRUE, the instance afterwards gets moved into the copy code (online change)
END_VAR
VAR
END_VAR
IF NOT bInCopyCode THEN
	SUPER^.CreateEx(Tc3_EventLogger.SUCCESS_EVENT, 0);
END_IF
END_METHOD

END_FUNCTION_BLOCK

// ---- POUs/Analytics/Analysis/Networks/N01 OEEStatus/FB_N1_OEEStatus.TcPOU
//Analytics Network "OEEStatus" with ID: 1
FUNCTION_BLOCK FB_N1_OEEStatus
VAR_OUTPUT
	bError: BOOL;
	ipTcResult: I_TcMessage := fbTcMsgSuccess;
END_VAR
VAR
	fbTcMsgSuccess: FB_TcMessageSuccess;
	
	//Modules
	fbM1_OverallEquipmentEffectivenessOEE: FB_N1_M1_OverallEquipmentEffectivenessOEE;
	fbM2_ProductionModeTimingAnalysis: FB_N1_M2_ProductionModeTimingAnalysis;
	fbM3_OEETrendLine: FB_N1_M3_OEETrendLine;
	fbM4_ProductionQuantityAnalysis: FB_N1_M4_ProductionQuantityAnalysis;
	fbM5_ProductivityInterval: FB_N1_M5_ProductivityInterval;
END_VAR

METHOD Call : BOOL
VAR_INPUT
	pAnalysis: POINTER TO FB_Analysis;
END_VAR
VAR
END_VAR

ValueMapping(pAnalysis);

//The Overall Equipment Effectiveness (OEE) algorithm calculates key values to compare the current manufacturing process with its full potential. Optional a boolean signal for Enable Execution can be selected, so that the algorithm is just active if the value of the selected signal is TRUE.
fbM1_OverallEquipmentEffectivenessOEE.tOperatingTime:= fbM2_ProductionModeTimingAnalysis.fbTimeOnTotal.nRaw;
fbM1_OverallEquipmentEffectivenessOEE.Call(pAnalysis^.nContext);

//The Timing Analysis 1Ch measures time difference between on- and off-periods and counts the amount of on-periods. The on-period starts when the condition of operator and threshold is met. Optional a boolean signal for Enable Execution can be selected, so that the algorithm is just active if the value of the selected signal is TRUE.
fbM2_ProductionModeTimingAnalysis.Call(pAnalysis^.nContext);

//This Module is used for the One-click Dashboard to generate a special analytics trend chart.
fbM3_OEETrendLine.fDataInCh1:= fbM1_OverallEquipmentEffectivenessOEE.fOEE;
fbM3_OEETrendLine.fDataInCh2:= fbM1_OverallEquipmentEffectivenessOEE.fAvailability;
fbM3_OEETrendLine.fDataInCh3:= fbM1_OverallEquipmentEffectivenessOEE.fPerformance;
fbM3_OEETrendLine.fDataInCh4:= fbM1_OverallEquipmentEffectivenessOEE.fQuality;
fbM3_OEETrendLine.Call(pAnalysis^.nContext);

//The Lifecycle Analysis 1Ch calculates the elapsed and the estimated remaining cycles of a device. The input channel should provide boolean values so that every switching procedure represents a cycle. Optional a boolean signal for Enable Execution can be selected, so that the algorithm is just active if the value of the selected signal is TRUE.
fbM4_ProductionQuantityAnalysis.Call(pAnalysis^.nContext);

//The Productivity interval 1Ch counts the amount of triggers within a timespan to calculate the productivity. Threfore the timespan is set by time inputs and the expected number of pieces is configured. Optional a boolean signal for Enable Execution can be selected, so that the algorithm is just active if the value of the selected signal is TRUE.
fbM5_ProductivityInterval.Call(pAnalysis^.nContext);


//Error Handling
IF fbM1_OverallEquipmentEffectivenessOEE.bError THEN
	bError:= TRUE;
	ipTcResult:= fbM1_OverallEquipmentEffectivenessOEE.ipTcResult;
ELSIF fbM2_ProductionModeTimingAnalysis.bError THEN
	bError:= TRUE;
	ipTcResult:= fbM2_ProductionModeTimingAnalysis.ipTcResult;
ELSIF fbM3_OEETrendLine.bError THEN
	bError:= TRUE;
	ipTcResult:= fbM3_OEETrendLine.ipTcResult;
ELSIF fbM4_ProductionQuantityAnalysis.bError THEN
	bError:= TRUE;
	ipTcResult:= fbM4_ProductionQuantityAnalysis.ipTcResult;
ELSIF fbM5_ProductivityInterval.bError THEN
	bError:= TRUE;
	ipTcResult:= fbM5_ProductivityInterval.ipTcResult;
ELSE
	bError:= FALSE;
	ipTcResult:= fbTcMsgSuccess;
END_IF
END_METHOD

METHOD Reset : BOOL
VAR
	bResult: BOOL := TRUE;
END_VAR
bResult:= bResult AND fbM1_OverallEquipmentEffectivenessOEE.Reset();
bResult:= bResult AND fbM2_ProductionModeTimingAnalysis.Reset();
bResult:= bResult AND fbM3_OEETrendLine.Reset();
bResult:= bResult AND fbM4_ProductionQuantityAnalysis.Reset();
bResult:= bResult AND fbM5_ProductivityInterval.Reset();
Reset:= bResult;
END_METHOD

METHOD PRIVATE ValueMapping : BOOL
VAR_INPUT
	pAnalysis: POINTER TO FB_Analysis;
END_VAR
VAR
END_VAR

//Module fbM1_OverallEquipmentEffectivenessOEE
fbM1_OverallEquipmentEffectivenessOEE.tTimestamp:= pAnalysis^.ipVirtualInputSource.tTimestamp;
fbM1_OverallEquipmentEffectivenessOEE.tScheduledTime:= pAnalysis^.ipVirtualInputSource.nV1_lScheduledTime;
fbM1_OverallEquipmentEffectivenessOEE.nUnitsProduced:= pAnalysis^.ipVirtualInputSource.nV1_uTotalCount;
fbM1_OverallEquipmentEffectivenessOEE.nDefectiveUnits:= pAnalysis^.ipVirtualInputSource.nV1_uDefectiveCount;


//Module fbM2_ProductionModeTimingAnalysis
fbM2_ProductionModeTimingAnalysis.tTimestamp:= pAnalysis^.ipVirtualInputSource.tTimestamp;
fbM2_ProductionModeTimingAnalysis.bDataIn:= pAnalysis^.ipVirtualInputSource.bV1_bProductionMode;


//Module fbM3_OEETrendLine
fbM3_OEETrendLine.tTimestamp:= pAnalysis^.ipVirtualInputSource.tTimestamp;

//Module fbM4_ProductionQuantityAnalysis
fbM4_ProductionQuantityAnalysis.nDataIn:= pAnalysis^.ipVirtualInputSource.nV1_uTotalCount;


//Module fbM5_ProductivityInterval
fbM5_ProductivityInterval.tTimestamp:= pAnalysis^.ipVirtualInputSource.tTimestamp;
fbM5_ProductivityInterval.bDataIn:= pAnalysis^.ipVirtualInputSource.bV1_bTest;
fbM5_ProductivityInterval.tTimeStart:= pAnalysis^.ipVirtualInputSource.nV1_lStartTime;
fbM5_ProductivityInterval.tTimeStop:= pAnalysis^.ipVirtualInputSource.nV1_lStopTime;
fbM5_ProductivityInterval.bEnableExecution:= pAnalysis^.ipVirtualInputSource.bV1_bConfigure;
fbM5_ProductivityInterval.bReset:= pAnalysis^.ipVirtualInputSource.bV1_bReset;
END_METHOD

END_FUNCTION_BLOCK

// ---- POUs/Analytics/Analysis/Networks/N01 OEEStatus/Modules/FB_N1_M1_OverallEquipmentEffectivenessOEE.TcPOU
//The Overall Equipment Effectiveness (OEE) algorithm calculates key values to compare the current manufacturing process with its full potential. Optional a boolean signal for Enable Execution can be selected, so that the algorithm is just active if the value of the selected signal is TRUE.
FUNCTION_BLOCK FB_N1_M1_OverallEquipmentEffectivenessOEE
VAR_INPUT
	tScheduledTime: LINT;
	tOperatingTime: LINT;
	nUnitsProduced: ULINT;
	nDefectiveUnits: ULINT;
	tTimestamp: ULINT;
	bEnableExecution: BOOL := TRUE;
	bReset: BOOL;
	bReconfigure: BOOL := TRUE;
END_VAR
VAR_INPUT PERSISTENT
	tIdealCycleTime: LTIME;
	fThresholdLevelOkWarning: LREAL;
	fThresholdLevelWarningAlarm: LREAL;
END_VAR
VAR_OUTPUT
	bError: BOOL;
	ipTcResult: I_TcMessage;
	bNewResult: BOOL;
	fOEE: LREAL;
	eOeeClass: E_ALY_Classification_3Cls;
	fAvailability: LREAL;
	fPerformance: LREAL;
	fQuality: LREAL;
	fbTimeOeeEventWarning: FB_ALY_DateTime;
	fbTimeOeeEventAlarm: FB_ALY_DateTime;
END_VAR
VAR
	
	R_TRIG_Reconfigure: R_TRIG;
	
	fbALY_OverallEquipmentEffectiveness: FB_ALY_OverallEquipmentEffectiveness;
END_VAR
VAR PERSISTENT
	bConfigured: BOOL;
END_VAR

METHOD Call : BOOL
VAR_INPUT
	nCurrentContext: DWORD;
END_VAR
VAR
END_VAR
IF NOT bConfigured THEN
	bConfigured:= TRUE;

	tIdealCycleTime:= LTIME#7s;
	fThresholdLevelOkWarning:= 90;
	fThresholdLevelWarningAlarm:= 75;

END_IF

R_TRIG_Reconfigure(CLK:= bReconfigure);
IF R_TRIG_Reconfigure.Q THEN
	fbALY_OverallEquipmentEffectiveness.Configure(tIdealCycleTime:= tIdealCycleTime, fThresholdLevelOkWarning:= fThresholdLevelOkWarning, fThresholdLevelWarningAlarm:= fThresholdLevelWarningAlarm);

	bReconfigure:= FALSE;
END_IF

IF bReset THEN
	Reset();
END_IF

IF bEnableExecution THEN
	IF F_HasContext(nCurrentContext, nContext) THEN
		fbALY_OverallEquipmentEffectiveness.SetChannelValue(nChannel:= 1, Input:= tScheduledTime);
		fbALY_OverallEquipmentEffectiveness.SetChannelValue(nChannel:= 2, Input:= tOperatingTime);
		fbALY_OverallEquipmentEffectiveness.SetChannelValue(nChannel:= 3, Input:= nUnitsProduced);
		fbALY_OverallEquipmentEffectiveness.SetChannelValue(nChannel:= 4, Input:= nDefectiveUnits);

		fbALY_OverallEquipmentEffectiveness.Call(tTimestamp:= tTimestamp);

		bNewResult:= fbALY_OverallEquipmentEffectiveness.bNewResult;
		fOEE:= fbALY_OverallEquipmentEffectiveness.fOEE;
		eOeeClass:= fbALY_OverallEquipmentEffectiveness.eOeeClass;
		fAvailability:= fbALY_OverallEquipmentEffectiveness.fAvailability;
		fPerformance:= fbALY_OverallEquipmentEffectiveness.fPerformance;
		fQuality:= fbALY_OverallEquipmentEffectiveness.fQuality;
		fbTimeOeeEventWarning:= fbALY_OverallEquipmentEffectiveness.fbTimeOeeEventWarning;
		fbTimeOeeEventAlarm:= fbALY_OverallEquipmentEffectiveness.fbTimeOeeEventAlarm;

		bError:= fbALY_OverallEquipmentEffectiveness.bError;
		ipTcResult:= fbALY_OverallEquipmentEffectiveness.ipResultMessage;
	END_IF
ELSE
	bNewResult:= FALSE;
END_IF
END_METHOD

METHOD Reset : BOOL
VAR
END_VAR
Reset:= fbALY_OverallEquipmentEffectiveness.Reset();

bNewResult:= fbALY_OverallEquipmentEffectiveness.bNewResult;
fOEE:= fbALY_OverallEquipmentEffectiveness.fOEE;
eOeeClass:= fbALY_OverallEquipmentEffectiveness.eOeeClass;
fAvailability:= fbALY_OverallEquipmentEffectiveness.fAvailability;
fPerformance:= fbALY_OverallEquipmentEffectiveness.fPerformance;
fQuality:= fbALY_OverallEquipmentEffectiveness.fQuality;
fbTimeOeeEventWarning:= fbALY_OverallEquipmentEffectiveness.fbTimeOeeEventWarning;
fbTimeOeeEventAlarm:= fbALY_OverallEquipmentEffectiveness.fbTimeOeeEventAlarm;

bError:= NOT Reset;
ipTcResult:= fbALY_OverallEquipmentEffectiveness.ipResultMessage;
END_METHOD

METHOD SetHMI : BOOL
VAR_INPUT
	nContent: DINT;
	pContent: PVOID;
	bHMIReinit: BOOL;
END_VAR
VAR
	pHMI_C1_OEE_Status: POINTER TO ST_HMI_C1_OEE_Status;
END_VAR
SetHMI:= FALSE;

CASE nContent OF
	1:
		pHMI_C1_OEE_Status:= pContent;

		IF bHMIReinit AND bConfigured THEN
			pHMI_C1_OEE_Status^.stHMI_C1_Ctrl4_Overall_Equipment_Effectiveness_OEE.fM1_fThresholdLevelOkWarning:= fThresholdLevelOkWarning;
			pHMI_C1_OEE_Status^.stHMI_C1_Ctrl4_Overall_Equipment_Effectiveness_OEE.fM1_fThresholdLevelWarningAlarm:= fThresholdLevelWarningAlarm;
			SetHMI:= TRUE;
		END_IF

		pHMI_C1_OEE_Status^.stHMI_C1_Ctrl4_Overall_Equipment_Effectiveness_OEE.fM1_fOEE:= fOEE;
		pHMI_C1_OEE_Status^.stHMI_C1_Ctrl4_Overall_Equipment_Effectiveness_OEE.fM1_fAvailability:= fAvailability;
		pHMI_C1_OEE_Status^.stHMI_C1_Ctrl4_Overall_Equipment_Effectiveness_OEE.fM1_fPerformance:= fPerformance;
		pHMI_C1_OEE_Status^.stHMI_C1_Ctrl4_Overall_Equipment_Effectiveness_OEE.fM1_fQuality:= fQuality;
		pHMI_C1_OEE_Status^.stHMI_C1_Ctrl4_Overall_Equipment_Effectiveness_OEE.eM1_eOeeClass:= eOeeClass;
END_CASE
END_METHOD

METHOD GetHMI : BOOL
VAR_INPUT
	nContent: DINT;
	pContent: PVOID;
END_VAR
VAR
	pHMI_C1_OEE_Status: POINTER TO ST_HMI_C1_OEE_Status;
END_VAR

CASE nContent OF
	1:
		//OEE_Status
		pHMI_C1_OEE_Status:= pContent;

		IF pHMI_C1_OEE_Status^.stHMI_C1_Ctrl4_Overall_Equipment_Effectiveness_OEE.bTrigReconfigure THEN
			pHMI_C1_OEE_Status^.stHMI_C1_Ctrl4_Overall_Equipment_Effectiveness_OEE.bTrigReconfigure:= FALSE;
			bReconfigure:= TRUE;

			fThresholdLevelOkWarning:= pHMI_C1_OEE_Status^.stHMI_C1_Ctrl4_Overall_Equipment_Effectiveness_OEE.fM1_fThresholdLevelOkWarning;
			fThresholdLevelWarningAlarm:= pHMI_C1_OEE_Status^.stHMI_C1_Ctrl4_Overall_Equipment_Effectiveness_OEE.fM1_fThresholdLevelWarningAlarm;
		END_IF
END_CASE

GetHMI:= bReconfigure;
END_METHOD

PROPERTY nContext : DWORD
GET
nContext:= E_VirtualInput.eContext_V1_VirtualInputSource;
END_GET
END_PROPERTY

END_FUNCTION_BLOCK

// ---- POUs/Analytics/[Helper]/Common/F_HasContext.TcPOU
FUNCTION F_HasContext : BOOL
VAR_INPUT
	nContext: DWORD;
	nSearchContext: DWORD;
END_VAR
VAR
END_VAR


F_HasContext:= (nContext > 0) AND (((nContext AND nSearchContext) > 0) OR (nSearchContext = E_DataSourceContext.eContext_Unknown));

END_FUNCTION

// ---- POUs/Analytics/Analysis/Networks/N01 OEEStatus/Modules/FB_N1_M2_ProductionModeTimingAnalysis.TcPOU
//The Timing Analysis 1Ch measures time difference between on- and off-periods and counts the amount of on-periods. The on-period starts when the condition of operator and threshold is met. Optional a boolean signal for Enable Execution can be selected, so that the algorithm is just active if the value of the selected signal is TRUE.
FUNCTION_BLOCK FB_N1_M2_ProductionModeTimingAnalysis
VAR_INPUT
	bDataIn: BOOL;
	tTimestamp: ULINT;
	bEnableExecution: BOOL := TRUE;
	bReset: BOOL;
	bReconfigure: BOOL := TRUE;
END_VAR
VAR_INPUT PERSISTENT
	stThresholdLevelOn: ST_ALY_Threshold;
	fTolerance: LREAL;
END_VAR
VAR_OUTPUT
	bError: BOOL;
	ipTcResult: I_TcMessage;
	bNewResult: BOOL;
	bIsOn: BOOL;
	nCountOn: ULINT;
	fbTimeCurrentInterval: FB_ALY_TimeSpan;
	fbTimeOnTotal: FB_ALY_TimeSpan;
	fbTimeOffTotal: FB_ALY_TimeSpan;
	fbTimeLastInterval: FB_ALY_TimeSpan;
END_VAR
VAR
	
	R_TRIG_Reconfigure: R_TRIG;
	
	fbALY_TimingAnalysis_1Ch: FB_ALY_TimingAnalysis_1Ch;
END_VAR
VAR PERSISTENT
	bConfigured: BOOL;
END_VAR

METHOD Call : BOOL
VAR_INPUT
	nCurrentContext: DWORD;
END_VAR
VAR
END_VAR
IF NOT bConfigured THEN
	bConfigured:= TRUE;

	fTolerance:= 0;

	stThresholdLevelOn.eComparisonOperator:= E_ALY_ComparisonOperator.GreaterThanOrEqualTo;
	stThresholdLevelOn.fThreshold:= 1;

	fbALY_TimingAnalysis_1Ch.fTolerance:= fTolerance;
END_IF

R_TRIG_Reconfigure(CLK:= bReconfigure);
IF R_TRIG_Reconfigure.Q THEN
	fbALY_TimingAnalysis_1Ch.ConfigureChannel(stThresholdLevel:= stThresholdLevelOn);

	fbALY_TimingAnalysis_1Ch.Configure();

	bReconfigure:= FALSE;
END_IF

IF bReset THEN
	Reset();
END_IF

IF bEnableExecution THEN
	IF F_HasContext(nCurrentContext, nContext) THEN
		fbALY_TimingAnalysis_1Ch.SetChannelValue(Input:= bDataIn);

		fbALY_TimingAnalysis_1Ch.Call(tTimestamp:= tTimestamp);

		bNewResult:= fbALY_TimingAnalysis_1Ch.bNewResult;
		bIsOn:= fbALY_TimingAnalysis_1Ch.bIsOn;
		nCountOn:= fbALY_TimingAnalysis_1Ch.nCountOn;
		fbTimeCurrentInterval:= fbALY_TimingAnalysis_1Ch.fbTimeCurrentInterval;
		fbTimeOnTotal:= fbALY_TimingAnalysis_1Ch.fbTimeOnTotal;
		fbTimeOffTotal:= fbALY_TimingAnalysis_1Ch.fbTimeOffTotal;
		fbTimeLastInterval:= fbALY_TimingAnalysis_1Ch.fbTimeLastInterval;

		bError:= fbALY_TimingAnalysis_1Ch.bError;
		ipTcResult:= fbALY_TimingAnalysis_1Ch.ipResultMessage;
	END_IF
ELSE
	bNewResult:= FALSE;
END_IF
END_METHOD

METHOD Reset : BOOL
VAR
END_VAR
Reset:= fbALY_TimingAnalysis_1Ch.Reset();

bNewResult:= fbALY_TimingAnalysis_1Ch.bNewResult;
bIsOn:= fbALY_TimingAnalysis_1Ch.bIsOn;
nCountOn:= fbALY_TimingAnalysis_1Ch.nCountOn;
fbTimeCurrentInterval:= fbALY_TimingAnalysis_1Ch.fbTimeCurrentInterval;
fbTimeOnTotal:= fbALY_TimingAnalysis_1Ch.fbTimeOnTotal;
fbTimeOffTotal:= fbALY_TimingAnalysis_1Ch.fbTimeOffTotal;
fbTimeLastInterval:= fbALY_TimingAnalysis_1Ch.fbTimeLastInterval;

bError:= NOT Reset;
ipTcResult:= fbALY_TimingAnalysis_1Ch.ipResultMessage;
END_METHOD

PROPERTY nContext : DWORD
GET
nContext:= E_VirtualInput.eContext_V1_VirtualInputSource;
END_GET
END_PROPERTY

END_FUNCTION_BLOCK

// ---- POUs/Analytics/Analysis/Networks/N01 OEEStatus/Modules/FB_N1_M3_OEETrendLine.TcPOU
//This Module is used for the One-click Dashboard to generate a special analytics trend chart.
FUNCTION_BLOCK FB_N1_M3_OEETrendLine
VAR_INPUT
	fDataInCh1: LREAL;
	fDataInCh2: LREAL;
	fDataInCh3: LREAL;
	fDataInCh4: LREAL;
	tTimestamp: ULINT;
	bEnableExecution: BOOL := TRUE;
	bReset: BOOL;
	aChannelNames: ARRAY [0..3] OF STRING(255);
END_VAR
VAR_OUTPUT
	bError: BOOL;
	ipTcResult: I_TcMessage;
	bNewResult: BOOL;
	fbLastValue: FB_ALY_DateTime;
END_VAR
VAR_OUTPUT PERSISTENT
	aTrendData: ARRAY [1..4] OF ARRAY [1..10080] OF LREAL;
	nCountValues: UDINT;
END_VAR
VAR
	
	bConfigured: BOOL;
	
	fbALY_TrendLine: FB_ALY_TrendLine(nNumChannels:=4);
END_VAR
VAR PERSISTENT
	nLastValueTimestamp: ULINT;
END_VAR

METHOD Call : BOOL
VAR_INPUT
	nCurrentContext: DWORD;
END_VAR
VAR
END_VAR
IF NOT bConfigured THEN
	bConfigured:= TRUE;

	aChannelNames[0]:= 'OEE ';
	aChannelNames[1]:= 'Availability';
	aChannelNames[2]:= 'Performance';
	aChannelNames[3]:= 'Quality';


	fbALY_TrendLine.SetChannelInitial(nChannel:=1, pArrayIn:= ADR(aTrendData[1]), nArrayInSize:= SIZEOF(aTrendData[1]));
	fbALY_TrendLine.SetChannelInitial(nChannel:=2, pArrayIn:= ADR(aTrendData[2]), nArrayInSize:= SIZEOF(aTrendData[2]));
	fbALY_TrendLine.SetChannelInitial(nChannel:=3, pArrayIn:= ADR(aTrendData[3]), nArrayInSize:= SIZEOF(aTrendData[3]));
	fbALY_TrendLine.SetChannelInitial(nChannel:=4, pArrayIn:= ADR(aTrendData[4]), nArrayInSize:= SIZEOF(aTrendData[4]));
	fbALY_TrendLine.SetInitial(tLastValue:= nLastValueTimestamp, nCountValues:= nCountValues);
END_IF

IF bReset THEN
	Reset();
END_IF

IF bEnableExecution THEN
	IF F_HasContext(nCurrentContext, nContext) THEN
		fbALY_TrendLine.SetChannelValue(nChannel:= 1, Input:= fDataInCh1);
		fbALY_TrendLine.SetChannelValue(nChannel:= 2, Input:= fDataInCh2);
		fbALY_TrendLine.SetChannelValue(nChannel:= 3, Input:= fDataInCh3);
		fbALY_TrendLine.SetChannelValue(nChannel:= 4, Input:= fDataInCh4);

		fbALY_TrendLine.Call(tTimestamp:= tTimestamp);

		bNewResult:= fbALY_TrendLine.bNewResult;
		fbLastValue:= fbALY_TrendLine.fbLastValue;
		nCountValues:= fbALY_TrendLine.nCountValues;

		bError:= fbALY_TrendLine.bError;
		ipTcResult:= fbALY_TrendLine.ipResultMessage;

		IF bNewResult THEN
			fbALY_TrendLine.GetChannelOutputArray(nChannel:=1, pArrayOut:= ADR(aTrendData[1]), nArrayOutSize:= SIZEOF(aTrendData[1]));
			fbALY_TrendLine.GetChannelOutputArray(nChannel:=2, pArrayOut:= ADR(aTrendData[2]), nArrayOutSize:= SIZEOF(aTrendData[2]));
			fbALY_TrendLine.GetChannelOutputArray(nChannel:=3, pArrayOut:= ADR(aTrendData[3]), nArrayOutSize:= SIZEOF(aTrendData[3]));
			fbALY_TrendLine.GetChannelOutputArray(nChannel:=4, pArrayOut:= ADR(aTrendData[4]), nArrayOutSize:= SIZEOF(aTrendData[4]));
		END_IF

		nLastValueTimestamp:= fbLastValue.nRaw;
	END_IF
ELSE
	bNewResult:= FALSE;
END_IF
END_METHOD

METHOD Reset : BOOL
VAR
END_VAR
Reset:= fbALY_TrendLine.Reset();

bNewResult:= fbALY_TrendLine.bNewResult;
fbLastValue:= fbALY_TrendLine.fbLastValue;
nCountValues:= fbALY_TrendLine.nCountValues;

bError:= NOT Reset;
ipTcResult:= fbALY_TrendLine.ipResultMessage;
END_METHOD

METHOD SetHMI : BOOL
VAR_INPUT
	nContent: DINT;
	pContent: PVOID;
	bHMIReinit: BOOL;
END_VAR
VAR
	pHMI_C1_OEE_Status: POINTER TO ST_HMI_C1_OEE_Status;
END_VAR
SetHMI:= FALSE;

CASE nContent OF
	1:
		pHMI_C1_OEE_Status:= pContent;


		pHMI_C1_OEE_Status^.stHMI_C1_Ctrl2_OEE_Trend_Line.aM3_aTrendData:= aTrendData;
		pHMI_C1_OEE_Status^.stHMI_C1_Ctrl2_OEE_Trend_Line.tM3_fbLastValue:= F_RawTimeToDCTimestruct(nRaw:= fbLastValue.nRaw, nUtcTimeBias:= -480);; //UTC Offset [(UTC+08:00) Kuala Lumpur, Singapore]
		pHMI_C1_OEE_Status^.stHMI_C1_Ctrl2_OEE_Trend_Line.nM3_nCountValues:= nCountValues;
		pHMI_C1_OEE_Status^.stHMI_C1_Ctrl2_OEE_Trend_Line.aM3_aChannelNames:= aChannelNames;
END_CASE

SetHMI:= TRUE;
END_METHOD

METHOD GetHMI : BOOL
VAR_INPUT
	nContent: DINT;
	pContent: PVOID;
END_VAR
VAR
END_VAR
END_METHOD

PROPERTY nContext : DWORD
GET
nContext:= E_VirtualInput.eContext_V1_VirtualInputSource;
END_GET
END_PROPERTY

END_FUNCTION_BLOCK

// ---- POUs/Analytics/[Helper]/Convert Timestamp/F_RawTimeToDCTimestruct.TcPOU
FUNCTION F_RawTimeToDCTimestruct : DCTimestruct
VAR_INPUT
	nRaw: ULINT;
	nUtcTimeBias: INT;
END_VAR
VAR
	fbTime: FB_ALY_DateTime;
END_VAR

fbTime.nRaw:= nRaw;
fbTime.nUtcTimeBias:= nUtcTimeBias;
F_RawTimeToDCTimestruct:= fbTime.stStructured;

END_FUNCTION

// ---- POUs/Analytics/Analysis/Networks/N01 OEEStatus/Modules/FB_N1_M4_ProductionQuantityAnalysis.TcPOU
//The Lifecycle Analysis 1Ch calculates the elapsed and the estimated remaining cycles of a device. The input channel should provide boolean values so that every switching procedure represents a cycle. Optional a boolean signal for Enable Execution can be selected, so that the algorithm is just active if the value of the selected signal is TRUE.
FUNCTION_BLOCK FB_N1_M4_ProductionQuantityAnalysis
VAR_INPUT
	nDataIn: ULINT;
	bEnableExecution: BOOL := TRUE;
	bReset: BOOL;
	bReconfigure: BOOL := TRUE;
END_VAR
VAR_INPUT PERSISTENT
	stThresholdEdge: ST_ALY_Threshold;
	nCyclesEstimated: ULINT;
	fTolerance: LREAL;
END_VAR
VAR_OUTPUT
	bError: BOOL;
	ipTcResult: I_TcMessage;
	bNewResult: BOOL;
	nCyclesElapsed: ULINT;
	nCyclesRemaining: LINT;
	bLifecyclesElapsed: BOOL;
END_VAR
VAR
	
	R_TRIG_Reconfigure: R_TRIG;
	
	fbALY_LifecycleAnalysis_1Ch: FB_ALY_LifecycleAnalysis_1Ch;
END_VAR
VAR PERSISTENT
	bConfigured: BOOL;
END_VAR

METHOD Call : BOOL
VAR_INPUT
	nCurrentContext: DWORD;
END_VAR
VAR
END_VAR
IF NOT bConfigured THEN
	bConfigured:= TRUE;

	nCyclesEstimated:= 1000;
	fTolerance:= 0;

	stThresholdEdge.eComparisonOperator:= E_ALY_ComparisonOperator.Equals;
	stThresholdEdge.fThreshold:= 1;

	fbALY_LifecycleAnalysis_1Ch.fTolerance:= fTolerance;
END_IF

R_TRIG_Reconfigure(CLK:= bReconfigure);
IF R_TRIG_Reconfigure.Q THEN
	fbALY_LifecycleAnalysis_1Ch.ConfigureChannel(stThresholdEdge:= stThresholdEdge);

	fbALY_LifecycleAnalysis_1Ch.Configure(nCyclesEstimated:= nCyclesEstimated);

	bReconfigure:= FALSE;
END_IF

IF bReset THEN
	Reset();
END_IF

IF bEnableExecution THEN
	IF F_HasContext(nCurrentContext, nContext) THEN
		fbALY_LifecycleAnalysis_1Ch.SetChannelValue(Input:= nDataIn);

		fbALY_LifecycleAnalysis_1Ch.Call();

		bNewResult:= fbALY_LifecycleAnalysis_1Ch.bNewResult;
		nCyclesElapsed:= fbALY_LifecycleAnalysis_1Ch.nCyclesElapsed;
		nCyclesRemaining:= fbALY_LifecycleAnalysis_1Ch.nCyclesRemaining;
		bLifecyclesElapsed:= fbALY_LifecycleAnalysis_1Ch.bLifecyclesElapsed;

		bError:= fbALY_LifecycleAnalysis_1Ch.bError;
		ipTcResult:= fbALY_LifecycleAnalysis_1Ch.ipResultMessage;
	END_IF
ELSE
	bNewResult:= FALSE;
END_IF
END_METHOD

METHOD Reset : BOOL
VAR
END_VAR
Reset:= fbALY_LifecycleAnalysis_1Ch.Reset();

bNewResult:= fbALY_LifecycleAnalysis_1Ch.bNewResult;
nCyclesElapsed:= fbALY_LifecycleAnalysis_1Ch.nCyclesElapsed;
nCyclesRemaining:= fbALY_LifecycleAnalysis_1Ch.nCyclesRemaining;
bLifecyclesElapsed:= fbALY_LifecycleAnalysis_1Ch.bLifecyclesElapsed;

bError:= NOT Reset;
ipTcResult:= fbALY_LifecycleAnalysis_1Ch.ipResultMessage;
END_METHOD

METHOD SetHMI : BOOL
VAR_INPUT
	nContent: DINT;
	pContent: PVOID;
	bHMIReinit: BOOL;
END_VAR
VAR
	pHMI_C1_OEE_Status: POINTER TO ST_HMI_C1_OEE_Status;
END_VAR
SetHMI:= FALSE;

CASE nContent OF
	1:
		pHMI_C1_OEE_Status:= pContent;

		IF bHMIReinit AND bConfigured THEN
			SetHMI:= TRUE;
		END_IF

		pHMI_C1_OEE_Status^.stHMI_C1_Ctrl1_Production_Quantity_Analysis.fM4_nCyclesElapsed:= TO_LREAL(nCyclesElapsed);
		pHMI_C1_OEE_Status^.stHMI_C1_Ctrl1_Production_Quantity_Analysis.fM4_nCyclesRemaining:= TO_LREAL(nCyclesRemaining);
END_CASE
END_METHOD

METHOD GetHMI : BOOL
VAR_INPUT
	nContent: DINT;
	pContent: PVOID;
END_VAR
VAR
	pHMI_C1_OEE_Status: POINTER TO ST_HMI_C1_OEE_Status;
END_VAR

CASE nContent OF
	1:
		//OEE_Status
		pHMI_C1_OEE_Status:= pContent;

		IF pHMI_C1_OEE_Status^.stHMI_C1_Ctrl1_Production_Quantity_Analysis.bTrigReconfigure THEN
			pHMI_C1_OEE_Status^.stHMI_C1_Ctrl1_Production_Quantity_Analysis.bTrigReconfigure:= FALSE;
			bReconfigure:= TRUE;

		END_IF
END_CASE

GetHMI:= bReconfigure;
END_METHOD

PROPERTY nContext : DWORD
GET
nContext:= E_VirtualInput.eContext_V1_VirtualInputSource;
END_GET
END_PROPERTY

END_FUNCTION_BLOCK

// ---- POUs/Analytics/Analysis/Networks/N01 OEEStatus/Modules/FB_N1_M5_ProductivityInterval.TcPOU
//The Productivity interval 1Ch counts the amount of triggers within a timespan to calculate the productivity. Threfore the timespan is set by time inputs and the expected number of pieces is configured. Optional a boolean signal for Enable Execution can be selected, so that the algorithm is just active if the value of the selected signal is TRUE.
FUNCTION_BLOCK FB_N1_M5_ProductivityInterval
VAR_INPUT
	bDataIn: BOOL;
	tTimeStart: LWORD;
	tTimeStop: LWORD;
	tTimestamp: ULINT;
	bEnableExecution: BOOL := TRUE;
	bReset: BOOL;
	bReconfigure: BOOL := TRUE;
END_VAR
VAR_INPUT PERSISTENT
	stThresholdEdge: ST_ALY_Threshold;
	nExpectedPieces: ULINT:=3840;
	fTolerance: LREAL;
END_VAR
VAR_OUTPUT
	bError: BOOL;
	ipTcResult: I_TcMessage;
	bNewResult: BOOL;
	bWithinInterval: BOOL;
	fbCurrentTimestamp: FB_ALY_DateTime;
	fbIntervalLength: FB_ALY_TimeSpan;
	fbElapsedTime: FB_ALY_TimeSpan;
	fbRemainingTime: FB_ALY_TimeSpan;
	nProducedInInterval: ULINT;
	nRemainingInInterval: ULINT;
	fCurrentProductivity: LREAL;
	fExpectedProductivity: LREAL;
	fLastFullPeriodProductivity: LREAL;
END_VAR
VAR
	
	R_TRIG_Reconfigure: R_TRIG;
	
	fbALY_ProductivityInterval_1Ch: FB_ALY_ProductivityInterval_1Ch := ( bPersistent:= TRUE );
END_VAR
VAR PERSISTENT
	bConfigured: BOOL;
END_VAR

METHOD Call : BOOL
VAR_INPUT
	nCurrentContext: DWORD;
END_VAR
VAR
END_VAR
IF NOT bConfigured THEN
	bConfigured:= TRUE;

	nExpectedPieces:= 1000;
	fTolerance:= 0;

	stThresholdEdge.eComparisonOperator:= E_ALY_ComparisonOperator.GreaterThanOrEqualTo;
	stThresholdEdge.fThreshold:= 1;

	fbALY_ProductivityInterval_1Ch.fTolerance:= fTolerance;
END_IF

R_TRIG_Reconfigure(CLK:= bReconfigure);
IF R_TRIG_Reconfigure.Q THEN
	fbALY_ProductivityInterval_1Ch.ConfigureChannel(stThresholdEdge:= stThresholdEdge);

	fbALY_ProductivityInterval_1Ch.Configure(nExpectedPieces:= nExpectedPieces);

	bReconfigure:= FALSE;
END_IF

IF bReset THEN
	Reset();
END_IF

IF bEnableExecution THEN
	IF F_HasContext(nCurrentContext, nContext) THEN
		fbALY_ProductivityInterval_1Ch.SetChannelValue(Input:= bDataIn);

		fbALY_ProductivityInterval_1Ch.Call(tTimeStart:= TO_LTIME(tTimeStart), tTimeStop:= TO_LTIME(tTimeStop), tTimestamp:= tTimestamp);

		bNewResult:= fbALY_ProductivityInterval_1Ch.bNewResult;
		bWithinInterval:= fbALY_ProductivityInterval_1Ch.bWithinInterval;
		fbCurrentTimestamp:= fbALY_ProductivityInterval_1Ch.fbCurrentTimestamp;
		fbIntervalLength:= fbALY_ProductivityInterval_1Ch.fbIntervalLength;
		fbElapsedTime:= fbALY_ProductivityInterval_1Ch.fbElapsedTime;
		fbRemainingTime:= fbALY_ProductivityInterval_1Ch.fbRemainingTime;
		nProducedInInterval:= fbALY_ProductivityInterval_1Ch.nProducedInInterval;
		nRemainingInInterval:= fbALY_ProductivityInterval_1Ch.nRemainingInInterval;
		fCurrentProductivity:= fbALY_ProductivityInterval_1Ch.fCurrentProductivity;
		fExpectedProductivity:= fbALY_ProductivityInterval_1Ch.fExpectedProductivity;
		fLastFullPeriodProductivity:= fbALY_ProductivityInterval_1Ch.fLastFullPeriodProductivity;

		bError:= fbALY_ProductivityInterval_1Ch.bError;
		ipTcResult:= fbALY_ProductivityInterval_1Ch.ipResultMessage;
	END_IF
ELSE
	bNewResult:= FALSE;
END_IF
END_METHOD

METHOD GetHMI : BOOL
VAR_INPUT
	nContent: DINT;
	pContent: PVOID;
END_VAR
VAR
	pHMI_C1_OEE_Status: POINTER TO ST_HMI_C1_OEE_Status;
END_VAR

CASE nContent OF
	1:
		//OEE_Status
		pHMI_C1_OEE_Status:= pContent;

		IF pHMI_C1_OEE_Status^.stHMI_C1_Ctrl3_Productivity_Interval.bTrigReconfigure THEN
			pHMI_C1_OEE_Status^.stHMI_C1_Ctrl3_Productivity_Interval.bTrigReconfigure:= FALSE;
			bReconfigure:= TRUE;

		END_IF
END_CASE

GetHMI:= bReconfigure;
END_METHOD

PROPERTY nContext : DWORD
GET
nContext:= E_VirtualInput.eContext_V1_VirtualInputSource;
END_GET
END_PROPERTY

METHOD Reset : BOOL
VAR
END_VAR
Reset:= fbALY_ProductivityInterval_1Ch.Reset();

bNewResult:= fbALY_ProductivityInterval_1Ch.bNewResult;
bWithinInterval:= fbALY_ProductivityInterval_1Ch.bWithinInterval;
fbCurrentTimestamp:= fbALY_ProductivityInterval_1Ch.fbCurrentTimestamp;
fbIntervalLength:= fbALY_ProductivityInterval_1Ch.fbIntervalLength;
fbElapsedTime:= fbALY_ProductivityInterval_1Ch.fbElapsedTime;
fbRemainingTime:= fbALY_ProductivityInterval_1Ch.fbRemainingTime;
nProducedInInterval:= fbALY_ProductivityInterval_1Ch.nProducedInInterval;
nRemainingInInterval:= fbALY_ProductivityInterval_1Ch.nRemainingInInterval;
fCurrentProductivity:= fbALY_ProductivityInterval_1Ch.fCurrentProductivity;
fExpectedProductivity:= fbALY_ProductivityInterval_1Ch.fExpectedProductivity;
fLastFullPeriodProductivity:= fbALY_ProductivityInterval_1Ch.fLastFullPeriodProductivity;

bError:= NOT Reset;
ipTcResult:= fbALY_ProductivityInterval_1Ch.ipResultMessage;
END_METHOD

METHOD SetHMI : BOOL
VAR_INPUT
	nContent: DINT;
	pContent: PVOID;
	bHMIReinit: BOOL;
END_VAR
VAR
	pHMI_C1_OEE_Status: POINTER TO ST_HMI_C1_OEE_Status;
END_VAR
SetHMI:= FALSE;

CASE nContent OF
	1:
		pHMI_C1_OEE_Status:= pContent;

		IF bHMIReinit AND bConfigured THEN
			SetHMI:= TRUE;
		END_IF

		pHMI_C1_OEE_Status^.stHMI_C1_Ctrl3_Productivity_Interval.fM5_nProducedInInterval:= TO_LREAL(nProducedInInterval);
		pHMI_C1_OEE_Status^.stHMI_C1_Ctrl3_Productivity_Interval.fM5_nRemainingInInterval:= TO_LREAL(nRemainingInInterval);
		pHMI_C1_OEE_Status^.stHMI_C1_Ctrl3_Productivity_Interval.tM5_fbElapsedTime:= fbElapsedTime.stStructured;
		pHMI_C1_OEE_Status^.stHMI_C1_Ctrl3_Productivity_Interval.tM5_fbRemainingTime:= fbRemainingTime.stStructured;
		pHMI_C1_OEE_Status^.stHMI_C1_Ctrl3_Productivity_Interval.fM5_fCurrentProductivity:= fCurrentProductivity;
		pHMI_C1_OEE_Status^.stHMI_C1_Ctrl3_Productivity_Interval.fM5_fExpectedProductivity:= fExpectedProductivity;
END_CASE
END_METHOD

END_FUNCTION_BLOCK

// ---- POUs/MAIN.TcPOU
PROGRAM MAIN
VAR
END_VAR

END_PROGRAM

// ---- POUs/Analytics/Sources/T1_InputSource/FB_T1_InputSource.TcPOU
FUNCTION_BLOCK FB_T1_InputSource IMPLEMENTS I_InputSource
VAR
	_eDataState: E_DataSourceState;
	
	_nElements: UDINT;
	_nCurrentElement: UDINT;
	_nDataHandle: ULINT;
	
	_nClientListHash: LWORD;
	_nCurrentClientHash: LWORD;
	
	_stInputs: ST_T1_Inputs;
	
	fbIotSymbol_GlobalVariables_bProductionMode: FB_ALYC_IotSymbol_BOOL := (stInitialConfig:= (sSymbolName:= 'GlobalVariables.bProductionMode'));
	fbIotSymbol_GlobalVariables_lScheduledTime: FB_ALYC_IotSymbol_LINT := (stInitialConfig:= (sSymbolName:= 'GlobalVariables.lScheduledTime'));
	fbIotSymbol_GlobalVariables_uProcessedCount: FB_ALYC_IotSymbol_ULINT := (stInitialConfig:= (sSymbolName:= 'GlobalVariables.uProcessedCount'));
	fbIotSymbol_GlobalVariables_nVisuProductCommand: FB_ALYC_IotSymbol_DINT := (stInitialConfig:= (sSymbolName:= 'GlobalVariables.nVisuProductCommand'));
	fbIotSymbol_GlobalVariables_uDefectiveCount: FB_ALYC_IotSymbol_ULINT := (stInitialConfig:= (sSymbolName:= 'GlobalVariables.uDefectiveCount'));
	fbIotSymbol_GlobalVariables_lStartTime: FB_ALYC_IotSymbol_LWORD := (stInitialConfig:= (sSymbolName:= 'GlobalVariables.lStartTime'));
	fbIotSymbol_GlobalVariables_lStopTime: FB_ALYC_IotSymbol_LWORD := (stInitialConfig:= (sSymbolName:= 'GlobalVariables.lStopTime'));
	fbIotSymbol_GlobalVariables_bConfigure: FB_ALYC_IotSymbol_BOOL := (stInitialConfig:= (sSymbolName:= 'GlobalVariables.bConfigure'));
	fbIotSymbol_GlobalVariables_bReset: FB_ALYC_IotSymbol_BOOL := (stInitialConfig:= (sSymbolName:= 'GlobalVariables.bReset'));
	fbIotSymbol_GlobalVariables_bTest: FB_ALYC_IotSymbol_BOOL := (stInitialConfig:= (sSymbolName:= 'GlobalVariables.bTest'));
	fbIotSymbol_GlobalVariables_uTotalCount: FB_ALYC_IotSymbol_ULINT := (stInitialConfig:= (sSymbolName:= 'GlobalVariables.uTotalCount'));
	
	//Target T1 = Broker:"127.0.0.1" Topic:"PackMLDemo/PlcStream1"
	fbStreamHelper: FB_ALYC_MqttStreamHelper := (nObjectID:= 16#01010010, nNumInputBuffer:= 20);
	bConfigured: BOOL := FALSE;
	
	fbTON_DataTimeout: TON;
END_VAR
VAR_STAT
	_nClientIndex: INT;
END_VAR

METHOD AddClient : BOOL
VAR_OUTPUT
	nClientID: LWORD;
END_VAR
VAR
END_VAR
nClientID:= TO_LWORD(EXPT(2,_nClientIndex));
_nClientIndex:= _nClientIndex + 1;

_nClientListHash:= _nClientListHash + nClientID;
END_METHOD

METHOD Call : BOOL
VAR
END_VAR

IF NOT bConfigured THEN
	//GlobalVariables.bProductionMode
	fbStreamHelper.AddIotSymbol(fbIotSymbol_GlobalVariables_bProductionMode);
	//GlobalVariables.lScheduledTime
	fbStreamHelper.AddIotSymbol(fbIotSymbol_GlobalVariables_lScheduledTime);
	//GlobalVariables.uProcessedCount
	fbStreamHelper.AddIotSymbol(fbIotSymbol_GlobalVariables_uProcessedCount);
	//GlobalVariables.nVisuProductCommand
	fbStreamHelper.AddIotSymbol(fbIotSymbol_GlobalVariables_nVisuProductCommand);
	//GlobalVariables.uDefectiveCount
	fbStreamHelper.AddIotSymbol(fbIotSymbol_GlobalVariables_uDefectiveCount);
	//GlobalVariables.lStartTime
	fbStreamHelper.AddIotSymbol(fbIotSymbol_GlobalVariables_lStartTime);
	//GlobalVariables.lStopTime
	fbStreamHelper.AddIotSymbol(fbIotSymbol_GlobalVariables_lStopTime);
	//GlobalVariables.bConfigure
	fbStreamHelper.AddIotSymbol(fbIotSymbol_GlobalVariables_bConfigure);
	//GlobalVariables.bReset
	fbStreamHelper.AddIotSymbol(fbIotSymbol_GlobalVariables_bReset);
	//GlobalVariables.bTest
	fbStreamHelper.AddIotSymbol(fbIotSymbol_GlobalVariables_bTest);
	//GlobalVariables.uTotalCount
	fbStreamHelper.AddIotSymbol(fbIotSymbol_GlobalVariables_uTotalCount);

	bConfigured:= TRUE;
END_IF

fbStreamHelper.Call();
IF fbStreamHelper.bError THEN
	_eDataState:= E_DataSourceState.eError;
ELSIF NOT fbStreamHelper.bConnected THEN
	_eDataState:= E_DataSourceState.eNotConnected;
ELSE
	_nElements:= fbStreamHelper.nNumElements;
	IF _nElements > 0 THEN
		_eDataState:= E_DataSourceState.eReceiveData;
	END_IF

	fbTON_DataTimeout(IN:= _nElements = 0, PT:= T#5S);
	IF fbTON_DataTimeout.Q THEN
		_eDataState:= E_DataSourceState.eWaitForData;
	END_IF
END_IF

IF _nElements > 0 THEN
	_nDataHandle:= _nDataHandle + 1;
	_nCurrentClientHash:= 0;
END_IF

_nCurrentElement:= 0;
END_METHOD

METHOD ClientDone : BOOL
VAR_INPUT
	nClientID: LWORD;
END_VAR
VAR
END_VAR
_nCurrentClientHash:=  _nCurrentClientHash + nClientID;
END_METHOD

METHOD GetData : BOOL
VAR_INPUT
	nElement: UDINT;
	pInputs: PVOID;
	nInputsSize: UDINT;
END_VAR
VAR_OUTPUT
	nTimestamp: ULINT;
	nContext: DWORD;
END_VAR
VAR
	_nElement: UDINT;
	_pInputs: PVOID;
	_nInputsSize: UDINT;
END_VAR
Analytics.fbT1_IecCriticalSection.Enter();

_nElement:= nElement;
_pInputs:= pInputs;
_nInputsSize:= nInputsSize;

nContext:= 0;
IF nElements > 0 THEN
	IF _nElement <= nElements THEN

		IF _nCurrentElement <> _nElement THEN

			//Set local raw inputs
			IF fbIotSymbol_GlobalVariables_bProductionMode.bVariableFound THEN
				_stInputs.bGlobalVariables_bProductionMode:= fbIotSymbol_GlobalVariables_bProductionMode.GetValue(_nElement);
			END_IF
			IF fbIotSymbol_GlobalVariables_lScheduledTime.bVariableFound THEN
				_stInputs.nGlobalVariables_lScheduledTime:= fbIotSymbol_GlobalVariables_lScheduledTime.GetValue(_nElement);
			END_IF
			IF fbIotSymbol_GlobalVariables_uProcessedCount.bVariableFound THEN
				_stInputs.nGlobalVariables_uProcessedCount:= fbIotSymbol_GlobalVariables_uProcessedCount.GetValue(_nElement);
			END_IF
			IF fbIotSymbol_GlobalVariables_nVisuProductCommand.bVariableFound THEN
				_stInputs.nGlobalVariables_nVisuProductCommand:= fbIotSymbol_GlobalVariables_nVisuProductCommand.GetValue(_nElement);
			END_IF
			IF fbIotSymbol_GlobalVariables_uDefectiveCount.bVariableFound THEN
				_stInputs.nGlobalVariables_uDefectiveCount:= fbIotSymbol_GlobalVariables_uDefectiveCount.GetValue(_nElement);
			END_IF
			IF fbIotSymbol_GlobalVariables_lStartTime.bVariableFound THEN
				_stInputs.nGlobalVariables_lStartTime:= fbIotSymbol_GlobalVariables_lStartTime.GetValue(_nElement);
			END_IF
			IF fbIotSymbol_GlobalVariables_lStopTime.bVariableFound THEN
				_stInputs.nGlobalVariables_lStopTime:= fbIotSymbol_GlobalVariables_lStopTime.GetValue(_nElement);
			END_IF
			IF fbIotSymbol_GlobalVariables_bConfigure.bVariableFound THEN
				_stInputs.bGlobalVariables_bConfigure:= fbIotSymbol_GlobalVariables_bConfigure.GetValue(_nElement);
			END_IF
			IF fbIotSymbol_GlobalVariables_bReset.bVariableFound THEN
				_stInputs.bGlobalVariables_bReset:= fbIotSymbol_GlobalVariables_bReset.GetValue(_nElement);
			END_IF
			IF fbIotSymbol_GlobalVariables_bTest.bVariableFound THEN
				_stInputs.bGlobalVariables_bTest:= fbIotSymbol_GlobalVariables_bTest.GetValue(_nElement);
			END_IF
			IF fbIotSymbol_GlobalVariables_uTotalCount.bVariableFound THEN
				_stInputs.nGlobalVariables_uTotalCount:= fbIotSymbol_GlobalVariables_uTotalCount.GetValue(_nElement);
			END_IF

			nContext:= E_DataSourceContext.eContext_10000;
			_nCurrentElement:= _nElement;
		END_IF

		//Set output values
		IF _pInputs > 0 THEN
			MEMCPY(_pInputs, ADR(_stInputs), _nInputsSize);
			nTimestamp:= fbStreamHelper.GetTimestampElement(_nElement);
		END_IF
	END_IF
	GetData:= TRUE;
ELSE
	GetData:= FALSE;
END_IF

Analytics.fbT1_IecCriticalSection.Leave();
END_METHOD

METHOD NewDataAvailable : BOOL
VAR_INPUT
	nLastDataHandle: ULINT;
END_VAR
VAR
END_VAR
NewDataAvailable:= _nElements > 0 AND _nDataHandle <> nLastDataHandle;
END_METHOD

PROPERTY eDataState : E_DataSourceState
GET
eDataState:= _eDataState;
END_GET
END_PROPERTY

PROPERTY bReadNewData : BOOL
GET
bReadNewData:= _nElements = 0 OR _nCurrentClientHash >= _nClientListHash;
END_GET
END_PROPERTY

PROPERTY nDataHandle : ULINT
GET
nDataHandle:= _nDataHandle;
END_GET
END_PROPERTY

PROPERTY nElements : UDINT
GET
nElements:= _nElements;
END_GET
END_PROPERTY

END_FUNCTION_BLOCK

// ---- POUs/Analytics/[Helper]/Common/FB_DataBuffer.TcPOU
FUNCTION_BLOCK FB_DataBuffer
VAR_OUTPUT
	nElements: UDINT;
END_VAR
VAR
	_nDataSize: UDINT;
	
	_pWriteBuffer: POINTER TO BYTE;
	_pWriteBufferTime: POINTER TO ARRAY [1..cEntryCount] OF ULINT;
	_pReadBuffer: POINTER TO BYTE;
	_pReadBufferTime: POINTER TO ARRAY [1..cEntryCount] OF ULINT;
	
	_pBuffer1: POINTER TO BYTE;
	_aBufferTime1: ARRAY [1..cEntryCount] OF ULINT;
	_pBuffer2: POINTER TO BYTE;
	_aBufferTime2: ARRAY [1..cEntryCount] OF ULINT;
	
	_nBufferIdx: INT := 1;
	
	_nBufferEntry_Add: UDINT;
	
	_bLock: BOOL;
	
END_VAR
VAR CONSTANT
	cEntryCount: UDINT := 25;
END_VAR

METHOD FB_init : BOOL
VAR_INPUT
	bInitRetains: BOOL; // if TRUE, the retain variables are initialized (warm start / cold start)
	bInCopyCode: BOOL; // if TRUE, the instance afterwards gets moved into the copy code (online change)
	nDataSize: UDINT;
END_VAR
VAR
END_VAR
IF NOT bInCopyCode THEN
	_nDataSize:= nDataSize;
	_Init();
END_IF
END_METHOD

METHOD FB_exit : BOOL
VAR_INPUT
	bInCopyCode: BOOL; // if TRUE, the exit method is called for exiting an instance that is copied afterwards (online change).
END_VAR
VAR
END_VAR
IF _pBuffer1 <> 0 THEN
	__DELETE(_pBuffer1);
END_IF

IF _pBuffer2 <> 0 THEN
	__DELETE(_pBuffer2);
END_IF

_pWriteBuffer:= 0;
_pWriteBufferTime:= 0;
_pReadBuffer:= 0;
_pReadBufferTime:= 0;

_nBufferIdx:= 0;
_nBufferEntry_Add:= 0;
END_METHOD

METHOD PRIVATE _Init : BOOL
VAR
END_VAR
IF _pBuffer1 <> 0 THEN
	__DELETE(_pBuffer1);
END_IF

IF _pBuffer2 <> 0 THEN
	__DELETE(_pBuffer2);
END_IF

_pBuffer1 := __NEW(BYTE, (_nDataSize * cEntryCount));
_pBuffer2 := __NEW(BYTE, (_nDataSize * cEntryCount));

_nBufferIdx:= 0;

Call();
END_METHOD

METHOD Call : BOOL
VAR
END_VAR
nElements:= 0;

IF TestAndSet(_bLock) THEN

	_nBufferIdx:= _nBufferIdx + 1;
	IF _nBufferIdx >= 3 THEN
		_nBufferIdx:= 1;
	END_IF

	CASE _nBufferIdx OF
		1:
			_pWriteBuffer:= _pBuffer1;
			_pReadBuffer:= _pBuffer2;

			_pWriteBufferTime:= ADR(_aBufferTime1);
			_pReadBufferTime:= ADR(_aBufferTime2);
		2:
			_pWriteBuffer:= _pBuffer2;
			_pReadBuffer:= _pBuffer1;

			_pWriteBufferTime:= ADR(_aBufferTime2);
			_pReadBufferTime:= ADR(_aBufferTime1);
	END_CASE

	nElements:= _nBufferEntry_Add;

	_nBufferEntry_Add:= 0;
	_bLock:= FALSE;
END_IF
END_METHOD

METHOD AddData : BOOL
VAR_INPUT
	pDataIn: PVOID;
END_VAR
VAR
END_VAR
IF TestAndSet(_bLock) THEN

	IF _pWriteBuffer <> 0 AND pDataIn <> 0 THEN

		IF _nBufferEntry_Add >= cEntryCount THEN
			_nBufferEntry_Add:= cEntryCount - 1;
		END_IF

		MEMCPY(_pWriteBuffer + (_nBufferEntry_Add * _nDataSize), pDataIn, _nDataSize);

		_nBufferEntry_Add:= _nBufferEntry_Add + 1;

		IF _pWriteBufferTime <> 0 THEN
			_pWriteBufferTime^[_nBufferEntry_Add]:= F_GetActualDcTime64();
		END_IF

	END_IF

	_bLock:= FALSE;
END_IF
END_METHOD

METHOD GetData : BOOL
VAR_INPUT
	nElement: UDINT(1..cEntryCount);
	pDataOut: PVOID;
END_VAR
VAR
END_VAR
IF nElement <= nElements THEN
	IF pDataOut <> 0 AND _pReadBuffer <> 0 THEN
		MEMCPY(pDataOut, _pReadBuffer + ((nElement-1) * _nDataSize), _nDataSize);
	END_IF
END_IF
END_METHOD

METHOD GetTimestamp : ULINT
VAR_INPUT
	nElement: UDINT(1..cEntryCount);
END_VAR
VAR
END_VAR
IF _pReadBufferTime <> 0 THEN
	GetTimestamp:= _pReadBufferTime^[nElement];
END_IF
END_METHOD

END_FUNCTION_BLOCK

// ---- POUs/Analytics/[Helper]/Common/FB_GetSampleIndex.TcPOU
FUNCTION_BLOCK FB_GetSampleIndex
VAR_INPUT
	nSample: UDINT;
	nOverSamplingFactor: UDINT;
	nMaxOverSampling: UDINT;
	nTimestamp: ULINT;
END_VAR
VAR_OUTPUT
	bNewIndex: BOOL;
	nIndex: UDINT;
END_VAR
VAR
	nIndexFactor: UDINT;
	nLastIndex: UDINT;
	nLastTimestamp: ULINT;
END_VAR


nIndex:= 1;

IF nOverSamplingFactor > 0 THEN
	nIndexFactor:= nMaxOverSampling / nOverSamplingFactor;

	IF nIndexFactor > 0 THEN
		nIndex:= (nSample - 1) / nIndexFactor;
		nIndex:= nIndex + 1;
	END_IF

	IF nIndex > nOverSamplingFactor THEN
		nIndex:= nOverSamplingFactor;
	END_IF
END_IF

bNewIndex:= nIndex <> nLastIndex OR nLastTimestamp <> nTimestamp;

nLastIndex:= nIndex;
nLastTimestamp:= nTimestamp;

END_FUNCTION_BLOCK

// ---- POUs/Analytics/[Helper]/Common/F_ANY_Negation.TcPOU
FUNCTION F_ANY_Negation : BOOL
VAR_INPUT
	Input: ANY;
END_VAR
VAR
	bReturn: BOOL;
	pREAL: POINTER TO REAL;
	pLREAL: POINTER TO LREAL;
	pBOOL: POINTER TO BOOL;
	pBYTE: POINTER TO BYTE;
	pINT: POINTER TO INT;
	pDINT: POINTER TO DINT;
	pLINT: POINTER TO LINT;
	pUINT: POINTER TO UINT;
	pUDINT: POINTER TO UDINT;
	pULINT: POINTER TO ULINT;
	pWORD: POINTER TO WORD;
	pDWORD: POINTER TO DWORD;
	pLWORD: POINTER TO LWORD;
END_VAR

IF input.pValue <> 0 THEN
	bReturn:= TRUE;

	CASE Input.TypeClass OF
		__SYSTEM.TYPE_CLASS.TYPE_REAL:
			pREAL:= input.pValue;
			pREAL^:= pREAL^ * -1;
		__SYSTEM.TYPE_CLASS.TYPE_LREAL:
			pLREAL:= input.pValue;
			pLREAL^:= pLREAL^ * -1;
		__SYSTEM.TYPE_CLASS.TYPE_BOOL:
			pBOOL:= input.pValue;
			pBOOL^:= NOT pBOOL^;
		__SYSTEM.TYPE_CLASS.TYPE_BYTE:
			pBYTE:= input.pValue;
			pBYTE^:= NOT pBYTE^;
		__SYSTEM.TYPE_CLASS.TYPE_INT:
			pINT:= input.pValue;
			pINT^:= pINT^ * -1;
		__SYSTEM.TYPE_CLASS.TYPE_DINT:
			pDINT:= input.pValue;
			pDINT^:= pDINT^ * -1;
		__SYSTEM.TYPE_CLASS.TYPE_LINT:
			pLINT:= input.pValue;
			pLINT^:= pLINT^ * -1;
		__SYSTEM.TYPE_CLASS.TYPE_UINT:
			pUINT:= input.pValue;
			pUINT^:= NOT pUINT^;
		__SYSTEM.TYPE_CLASS.TYPE_UDINT:
			pUDINT:= input.pValue;
			pUDINT^:= NOT pUDINT^;
		__SYSTEM.TYPE_CLASS.TYPE_ULINT:
			pULINT:= input.pValue;
			pULINT^:= NOT pULINT^;
		__SYSTEM.TYPE_CLASS.TYPE_WORD:
			pWORD:= input.pValue;
			pWORD^:= NOT pWORD^;
		__SYSTEM.TYPE_CLASS.TYPE_DWORD:
			pDWORD:= input.pValue;
			pDWORD^:= NOT pDWORD^;
		__SYSTEM.TYPE_CLASS.TYPE_LWORD:
			pLWORD:= input.pValue;
			pLWORD^:= NOT pLWORD^;
		ELSE
			bReturn:= FALSE;
	END_CASE
END_IF

F_ANY_Negation:= bReturn;

END_FUNCTION

// ---- POUs/Analytics/[Helper]/Common/F_ARRAY_To_LREAL_ARRAY.TcPOU
FUNCTION F_ARRAY_To_LREAL_ARRAY : BOOL
VAR_INPUT
	pDataIn: POINTER TO BYTE;
	cbDataIn: UDINT;
	eDataType: E_DTType;
END_VAR
VAR_IN_OUT
	aDataOut: ARRAY [*] OF LREAL;
END_VAR
VAR
	i: DINT;
	nPos: UDINT;
	
	pBOOL: POINTER TO BOOL;
	pBYTE: POINTER TO BYTE;
	pWORD: POINTER TO WORD;
	pDWORD: POINTER TO DWORD;
	pSINT: POINTER TO SINT;
	pUSINT: POINTER TO USINT;
	pINT: POINTER TO INT;
	pUINT: POINTER TO UINT;
	pDINT: POINTER TO DINT;
	pUDINT: POINTER TO UDINT;
	pLINT: POINTER TO LINT;
	pULINT: POINTER TO ULINT;
	pREAL: POINTER TO REAL;
	pLREAL: POINTER TO LREAL;
	pLWORD: POINTER TO LWORD;
END_VAR

FOR i := LOWER_BOUND(aDataOut,1) TO UPPER_BOUND(aDataOut,1) DO
	CASE eDataType OF
		E_DTType.NotInitialized:
			F_ARRAY_To_LREAL_ARRAY:= FALSE;
			RETURN;
		E_DTType.BOOL_:
			IF (nPos * 1) < cbDataIn THEN
				pBOOL:= pDataIn + (nPos * 1);
				aDataOut[i] := TO_LREAL(pBOOL^);
			END_IF
		E_DTType.BYTE_:
			IF (nPos * 1) < cbDataIn THEN
				pBYTE:= pDataIn + (nPos * 1);
				aDataOut[i] := TO_LREAL(pBYTE^);
			END_IF
		E_DTType.WORD_:
			IF (nPos * 2) < cbDataIn THEN
				pWORD:= pDataIn + (nPos * 2);
				aDataOut[i] := TO_LREAL(pWORD^);
			END_IF
		E_DTType.DWORD_:
			IF (nPos * 4) < cbDataIn THEN
				pDWORD:= pDataIn + (nPos * 4);
				aDataOut[i] := TO_LREAL(pDWORD^);
			END_IF
		E_DTType.SINT_:
			IF (nPos * 1) < cbDataIn THEN
				pSINT:= pDataIn + (nPos * 1);
				aDataOut[i] := TO_LREAL(pSINT^);
			END_IF
		E_DTType.INT_:
			IF (nPos * 2) < cbDataIn THEN
				pINT:= pDataIn + (nPos * 2);
				aDataOut[i] := TO_LREAL(pINT^);
			END_IF
		E_DTType.UINT_:
			IF (nPos * 2) < cbDataIn THEN
				pUINT:= pDataIn + (nPos * 2);
				aDataOut[i] := TO_LREAL(pUINT^);
			END_IF
		E_DTType.DINT_:
			IF (nPos * 4) < cbDataIn THEN
				pDINT:= pDataIn + (nPos * 4);
				aDataOut[i] := TO_LREAL(pDINT^);
			END_IF
		E_DTType.UDINT_:
			IF (nPos * 4) < cbDataIn THEN
				pUDINT:= pDataIn + (nPos * 4);
				aDataOut[i] := TO_LREAL(pUDINT^);
			END_IF
		E_DTType.LINT_:
			IF (nPos * 8) < cbDataIn THEN
				pLINT:= pDataIn + (nPos * 8);
				aDataOut[i] := TO_LREAL(pLINT^);
			END_IF
		E_DTType.ULINT_:
			IF (nPos * 8) < cbDataIn THEN
				pULINT:= pDataIn + (nPos * 8);
				aDataOut[i] := TO_LREAL(pULINT^);
			END_IF
		E_DTType.REAL_:
			IF (nPos * 4) < cbDataIn THEN
				pREAL:= pDataIn + (nPos * 4);
				aDataOut[i] := TO_LREAL(pREAL^);
			END_IF
		E_DTType.LREAL_:
			IF (nPos * 8) < cbDataIn THEN
				pLREAL:= pDataIn + (nPos * 8);
				aDataOut[i] := TO_LREAL(pLREAL^);
			END_IF
		E_DTType.LWORD_:
			IF (nPos * 8) < cbDataIn THEN
				pLWORD:= pDataIn + (nPos * 8);
				aDataOut[i] := TO_LREAL(pLWORD^);
			END_IF
	END_CASE

	nPos:= nPos + 1;
END_FOR

F_ARRAY_To_LREAL_ARRAY:= TRUE;

END_FUNCTION

// ---- POUs/Analytics/[Helper]/Common/F_ToANY.TcPOU
FUNCTION F_ToANY : __SYSTEM.AnyType
VAR_INPUT
	Input: ANY;
END_VAR
VAR
END_VAR

F_ToANY:= Input;

END_FUNCTION

// ---- POUs/Analytics/[Helper]/Convert Timestamp/F_AlyTimestampToFileTime.TcPOU
FUNCTION F_AlyTimestampToFileTime : ULINT
VAR_INPUT
	tTimestamp: ULINT;
END_VAR
VAR
	tFileTime: T_FILETIME;
	
	fbToUTC: FB_TzSpecificLocalTimeToFileTime;
	//Malay Peninsula Daylight Time
	//(UTC+08:00) Kuala Lumpur, Singapore
	tzInfo: ST_TimeZoneInformation := (bias := -480);
END_VAR

tFileTime:= DCTIME64_TO_Filetime(tTimestamp);

fbToUTC(in:= tFileTime, tzInfo:= tzInfo);
F_AlyTimestampToFileTime:= ULARGE_TO_ULINT(ULARGE_INTEGER(fbToUTC.out.dwHighDateTime, fbToUTC.out.dwLowDateTime));

END_FUNCTION

// ---- POUs/Analytics/[Helper]/Convert Timestamp/F_AlyTimestampToLocalTime.TcPOU
FUNCTION F_AlyTimestampToLocalTime : ULINT
VAR_INPUT
	tTimestamp: ULINT;
END_VAR
VAR
	tFileTime: T_FILETIME;
END_VAR

tFileTime:= DCTIME64_TO_Filetime(tTimestamp);
F_AlyTimestampToLocalTime:= ULARGE_TO_ULINT(ULARGE_INTEGER(tFileTime.dwHighDateTime, tFileTime.dwLowDateTime));

END_FUNCTION

// ---- POUs/Analytics/[Helper]/Convert Timestamp/F_DCTimestructToFileTime.TcPOU
FUNCTION F_DCTimestructToFileTime : ULINT
VAR_INPUT
	dtTimestamp: DCTIMESTRUCT;
END_VAR
VAR
	dcTime: T_DCTIME64;
END_VAR

dcTime:= DCTIMESTRUCT_TO_DCTIME64(dtTimestamp);
F_DCTimestructToFileTime:= F_AlyTimestampToFileTime(dcTime);

END_FUNCTION

// ---- POUs/Analytics/[Helper]/Convert Timestamp/F_FileTimeToDCTimestruct.TcPOU
FUNCTION F_FileTimeToDCTimestruct : DCTIMESTRUCT
VAR_INPUT
	tTimestamp: ULINT;
END_VAR
VAR
	tULarge: T_ULARGE_INTEGER;
	tFileTime: T_FILETIME;
	newDCTime: T_DCTIME64;
	
	fbToLocal: FB_FileTimeToTzSpecificLocalTime;
	//Malay Peninsula Daylight Time
	//(UTC+08:00) Kuala Lumpur, Singapore
	tzInfo: ST_TimeZoneInformation := (bias := -480);
END_VAR

tULarge:= ULINT_TO_ULARGE(tTimestamp);
tFileTime.dwLowDateTime:= tULarge.dwLowPart;
tFileTime.dwHighDateTime:= tULarge.dwHighPart;

fbToLocal(in:= tFileTime, tzInfo:= tzInfo);
newDCTime:= FILETIME_TO_DCTIME64(fbToLocal.out);

F_FileTimeToDCTimestruct:= DCTIME64_TO_DCTIMESTRUCT(newDCTime);

END_FUNCTION

// ---- POUs/Analytics/[Helper]/F_SampleTimeCheck.TcPOU
FUNCTION F_SampleTimeCheck : BOOL
VAR_INPUT
	nSampleTimestamp: ULINT;
	nLastSampleTimestamp: ULINT;
	nSampleTime: UDINT;
END_VAR
VAR
	nDeviation: UDINT := 500000; //Allowed deviation 0.5ms
END_VAR

IF nLastSampleTimestamp = 0 THEN
	F_SampleTimeCheck:= TRUE;
ELSIF nSampleTimestamp >= (nLastSampleTimestamp + (nSampleTime + nDeviation)) THEN
	F_SampleTimeCheck:= TRUE;
ELSIF nSampleTimestamp >= (nLastSampleTimestamp + (nSampleTime - nDeviation)) THEN
	F_SampleTimeCheck:= TRUE;
ELSE
	F_SampleTimeCheck:= FALSE;
END_IF

END_FUNCTION
